// Communicating Units-------------------------------------------------------
      L     DB1715.DBD   10;
      L     DB1715.DBD  106;
      ==D   ;
      =     #ComCIP;

// emergency OK -------------------------------------------------------------
      A     DB1715.DBX   75.0; //General Emergency Stop OK
      =     #EStopOK;

NETWORK
TITLE =read other unit's data

      SET   ;

// ... General Unit ----------/

      CALL FC   563 (
           ActReq                   := M    101.0,
           PLCNo                    := DB1715.DBW   14,
           SourceUnitNo             := 99,
           IsTUnit                  := FALSE,
           DstComDRec               := DB1715.GEN,
           RET_VAL                  := #wRetVal);

// ... CIP Unit ------------- /
      L     DB1711.DBD   46; // Select
      L     L#0; // Off
      ==D   ;
      JC    ELS1;
      TAK   ;
      L     DB1915.DBD   10; // CIP 1
      ==D   ;
      JC    M101;
      TAK   ;
      L     DB1925.DBD   10; // CIP 2
      ==D   ;
      JC    M102;
      TAK   ;
      L     DB1935.DBD   10; // CIP 3
      ==D   ;
      JC    M103;
      JU    ELS1;
M101: NOP   0; // Do 1
      CALL FC   563 (
           ActReq                   := M    101.0,
           PLCNo                    := 3,
           SourceUnitNo             := 91,
           IsTUnit                  := FALSE,
           DstComDRec               := DB1715.CIP,
           RET_VAL                  := #wRetVal);

      JU    FIN1;
M102: NOP   0; // Do 2
      CALL FC   563 (
           ActReq                   := M    101.0,
           PLCNo                    := 3,
           SourceUnitNo             := 92,
           IsTUnit                  := FALSE,
           DstComDRec               := DB1715.CIP,
           RET_VAL                  := #wRetVal);

      JU    FIN1;
M103: NOP   0; // Do 3
      CALL FC   563 (
           ActReq                   := M    101.0,
           PLCNo                    := 3,
           SourceUnitNo             := 93,
           IsTUnit                  := FALSE,
           DstComDRec               := DB1715.CIP,
           RET_VAL                  := #wRetVal);

      JU    FIN1;
ELS1: L     0;
      T     #iTmp;
      CALL SFC   21 (
           BVAL                     := #iTmp,
           RET_VAL                  := #iRetVal,
           BLK                      := DB1715.CIP);

FIN1: NOP   0;

NETWORK
TITLE =remote start
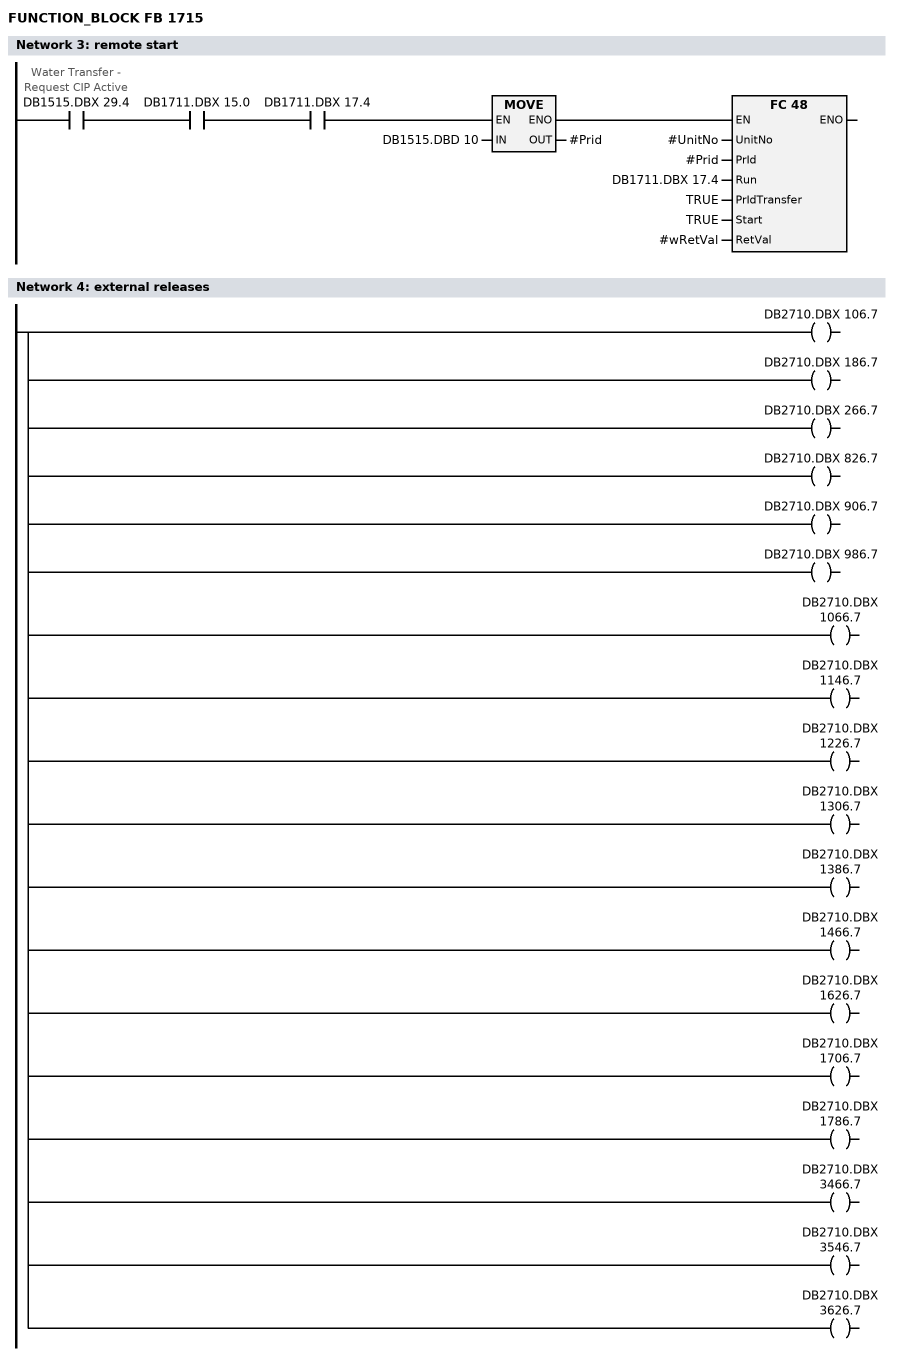

      SET   ;
      A     DB1515.DBX   29.4; // Water Transfer - Request CIP Active
      A     DB1711.DBX   15.0;
      A     DB1711.DBX   17.4;

      JCN   Strt;
      L     DB1515.DBD   10;
      T     #Prid;

      CALL FC    48 (
           UnitNo                   := #UnitNo,
           PrId                     := #Prid,
           Run                      := DB1711.DBX   17.4,
           PrIdTransfer             := TRUE,
           Start                    := TRUE,
           RetVal                   := #wRetVal);
Strt: NOP   0;
NETWORK
TITLE =external releases

      SET   ;
      =     DB2710.DBX  106.7;
      =     DB2710.DBX  186.7;
      =     DB2710.DBX  266.7;
      =     DB2710.DBX  826.7;
      =     DB2710.DBX  906.7;
      =     DB2710.DBX  986.7;
      =     DB2710.DBX 1066.7;
      =     DB2710.DBX 1146.7;
      =     DB2710.DBX 1226.7;
      =     DB2710.DBX 1306.7;
      =     DB2710.DBX 1386.7;
      =     DB2710.DBX 1466.7;
      =     DB2710.DBX 1626.7;
      =     DB2710.DBX 1706.7;
      =     DB2710.DBX 1786.7;
      =     DB2710.DBX 3466.7;
      =     DB2710.DBX 3546.7;
      =     DB2710.DBX 3626.7;
NETWORK
TITLE =write own unit data

      SET   ;

//-- CIP Communication ---------------------------------------
      AN    DB1711.DBX   15.0;
      AN    DB1711.DBX 1233.6; // CIP Active (Slave)
      A     #ComCIP;
      JCN   NCIP;
//Conductivity CIP Return
      L     DB1715.DBD  150;
      T     DB1711.DBD  626;

//Temperature CIP Return
      L     DB1715.DBD  146;
      T     DB1711.DBD  594;

//CIP Prerun Pump SP

      CALL FC    45 (
           SFM                      := DB1711.DBD  686,
           Indexes                  := #SFM36);


      L     0.000000e+000;
      A     #SFM36.I01;
      =     DB1715.DBX  171.7;
      JCN   pfc;
      L     DB1711.DBD  654;
pfc:  NOP   0;
      A     #SFM36.I02;
      =     DB1715.DBX  172.0;
      JCN   ppc;
      L     DB1711.DBD  670;
ppc:  NOP   0;
      A     #SFM36.I03;
      =     DB1715.DBX  171.6;
      JCN   pxc;
      L     DB1711.DBD  574;
pxc:  NOP   0;
      T     DB1715.DBD  182;

//CIP Return
      L     DB1711.DBD  558;
      T     DB1715.DBD  186;
      L     DB1715.DBD  138;
      T     DB1711.DBD  562;

//CIP Prerun
      L     DB1711.DBD  542;
      T     DB1715.DBD  190;
      L     DB1715.DBD  142;
      T     DB1711.DBD  546;

// Write Own Data to CIP
      L     DB1715.DBD   10;
      T     DB1715.DBD  154;

      L     DB1715.DBW   14;
      T     DB1715.DBW  158;

      L     DB1715.DBW   16;
      T     DB1715.DBW  160;

      L     DB1715.DBW   18;
      T     DB1715.DBW  162;

      L     DB1715.DBW   20;
      T     DB1715.DBW  164;

      L     DB1715.DBW   22;
      T     DB1715.DBW  166;

      A     DB1715.DBX   24.0;
      =     DB1715.DBX  168.0;

      A     DB1715.DBX   24.1;
      =     DB1715.DBX  168.1;

      A     DB1715.DBX   24.2;
      =     DB1715.DBX  168.2;

      A     DB1715.DBX   24.3;
      =     DB1715.DBX  168.3;

      A     DB1715.DBX   24.4;
      =     DB1715.DBX  168.4;

      A     DB1715.DBX   24.5;
      =     DB1715.DBX  168.5;

      A     DB1715.DBX   24.6;
      =     DB1715.DBX  168.6;

      A     DB1715.DBX   24.7;
      =     DB1715.DBX  168.7;

// Copy Data to CIP
      CALL SFC   20 (
           SRCBLK                   := DB1715.ToCIP,
           RET_VAL                  := #iRetVal,
           DSTBLK                   := DB1715.ToCIP);

NCIP: NOP   0;

//Empty Signal
//A     "U071SpID".SpI.Sig //!!!! Insert correct Empty Signal !!!
      CLR   ;
      =     DB1715.DBX   26.5;

//Full Signal
//A     "U071SpID".SpI.Sig //!!!! Insert correct Full Signal !!!
      CLR   ;
      =     DB1715.DBX   26.2;

//CIP Program Selected
      A     #CIP;
      =     DB1715.DBX   27.1;

// Emergency Stop
      A     #EStopOK; //If needed add or replace with own SpI
      =     DB1715.DBX   27.0; //Emergency Stop OK


NETWORK
TITLE =Signals to Filler / Mixer

// Watchdog
      A     M    100.7;
//    =     "F11_Watchdog"
//    =     "A11_Mixer_Watchdog"

      CLR   ;


END_FUNCTION_BLOCK

FUNCTION_BLOCK FB 1719
TITLE =U071: Packaging Plant 11
AUTHOR : Woermann
FAMILY : BOTEC_F1
NAME : Sim
VERSION : 0.1


VAR_TEMP
  CIP : BOOL ;	//CIP active
  xTmp : BOOL ;	//Temporary BOOL (free for general use)
  iTmp : INT ;	//Temporary INT (free for general use)
  rTmp : REAL ;	//Temporary REAL (free for general use)
  UnitNo : INT ;	//Unit Number
END_VAR
BEGIN
NETWORK
TITLE =General

      SET   ;
// get unit number ----------------------------------------------------------
      L     DB1710.DBW    0;
      T     #UnitNo;

// CIP ----------------------------------------------------------------------
      L     DB1711.DBD   54;
      L     0;
      <D    ;
      =     #CIP;

NETWORK
TITLE =Actuator

      A     DB1711.DBX   17.3;
      =     DB2710.DBX  105.3;
      =     DB2710.DBX  185.3;
      =     DB2710.DBX  265.3;
      =     DB2710.DBX  825.3;
      =     DB2710.DBX  905.3;
      =     DB2710.DBX  985.3;
      =     DB2710.DBX 1065.3;
      =     DB2710.DBX 1145.3;
      =     DB2710.DBX 1225.3;
      =     DB2710.DBX 1305.3;
      =     DB2710.DBX 1385.3;
      =     DB2710.DBX 1465.3;
      =     DB2710.DBX 1625.3;
      =     DB2710.DBX 1705.3;
      =     DB2710.DBX 1785.3;
      =     DB2710.DBX 3465.3;
      =     DB2710.DBX 3545.3;
      =     DB2710.DBX 3625.3;

NETWORK
TITLE =Special Input

      A     DB1711.DBX   17.3;
      =     DB2711.DBX  141.3;
      =     DB2711.DBX  201.3;
      =     DB2711.DBX  261.3;
      =     DB2711.DBX  321.3;
      =     DB2711.DBX  381.3;
      =     DB2711.DBX  681.3;
      =     DB2711.DBX  741.3;

NETWORK
TITLE =Counter

      A     DB1711.DBX   17.3;
      A     M    101.0;


      CLR   ;
NETWORK
TITLE =Analog Input

      A     DB1711.DBX   17.3;

NETWORK
TITLE =Universal Value

      A     DB1711.DBX   17.3;
//      =     "U071UnVD".unv001.Sim;
//      =     "U071UnVD".unv002.Sim;
//      =     "U071UnVD".unv003.Sim;
//      =     "U071UnVD".unv004.Sim;

NETWORK
TITLE =PID

      A     DB1711.DBX   17.3;

NETWORK
TITLE =Message

      A     DB1711.DBX   17.3;
//      =     "U071MsgD".msg001.Sim;
//      =     "U071MsgD".msg002.Sim;
//      =     "U071MsgD".msg003.Sim;

NETWORK
TITLE =VLT

      A     DB1711.DBX   17.3;

END_FUNCTION_BLOCK

FUNCTION_BLOCK FB 1725
TITLE =U072: Packaging Plant 12
FAMILY : BOTEC_F1
NAME : Comm
VERSION : 0.1


VAR_TEMP
  iRetVal : INT ;	//return value as integer
  wRetVal : WORD ;	//return value as word
  Run : BOOL ;	//Unit in "RUN" mode
  EStopOK : BOOL ;	//Emergency Stop OK
  CIP : BOOL ;	//CIP Program Selected
  ComCIP : BOOL ;	//Communication with CIP Active
  xTmp : BOOL ;	//Temporary BOOL (free for general use)
  iTmp : INT ;	//Temporary INT (free for general use)
  rTmp : REAL ;	//Temporary REAL (free for general use)
  dTmp : DINT ;	//Temporary DINT (free for general use)
  UnitNo : INT ;	//Unit Number
  EquipmentID : INT ;	//Equipment ID
  Prid : DINT ;	//Process ID
  SFM36 : STRUCT 	// CIP Pump Mode
   I00 : BOOL ;	// Off
   I01 : BOOL ;	// Flow
   I02 : BOOL ;	// Pressure
   I03 : BOOL ;	// Fix Speed
   I04 : BOOL ;
   I05 : BOOL ;
   I06 : BOOL ;
   I07 : BOOL ;
   I08 : BOOL ;
   I09 : BOOL ;
   I10 : BOOL ;
   I11 : BOOL ;
   I12 : BOOL ;
   I13 : BOOL ;
   I14 : BOOL ;
   I15 : BOOL ;
   I16 : BOOL ;
   I17 : BOOL ;
   I18 : BOOL ;
   I19 : BOOL ;
   I20 : BOOL ;
   I21 : BOOL ;
   I22 : BOOL ;
   I23 : BOOL ;
   I24 : BOOL ;
   I25 : BOOL ;
   I26 : BOOL ;
   I27 : BOOL ;
   I28 : BOOL ;
   I29 : BOOL ;
   I30 : BOOL ;
   I31 : BOOL ;
  END_STRUCT ;
END_VAR
BEGIN
NETWORK
TITLE =general

      SET   ;

// unit & equipment number ---------------------------------------------------
      L     DB1720.DBW    0;
      T     #UnitNo;

      L     DB1725.DBW   14;
      L     1000;
      *I    ;
      L     #UnitNo;
      +I    ;
      T     #EquipmentID;

// CIP ----------------------------------------------------------------------
      L     DB1725.DBW   18;
      L     0;
      <I    ;
      =     #CIP;

// Communicating Units-------------------------------------------------------
      L     DB1725.DBD   10;
      L     DB1725.DBD  106;
      ==D   ;
      =     #ComCIP;

// emergency OK -------------------------------------------------------------
      A     DB1725.DBX   75.0; //General Emergency Stop OK
      =     #EStopOK;

NETWORK
TITLE =read other unit's data

      SET   ;

// ... General Unit ----------/

      CALL FC   563 (
           ActReq                   := M    101.0,
           PLCNo                    := DB1725.DBW   14,
           SourceUnitNo             := 99,
           IsTUnit                  := FALSE,
           DstComDRec               := DB1725.GEN,
           RET_VAL                  := #wRetVal);


// ... CIP Unit ------------- /
      L     DB1721.DBD   46; // Select
      L     L#0; // Off
      ==D   ;
      JC    ELS1;
      TAK   ;
      L     DB1915.DBD   10; // CIP 1
      ==D   ;
      JC    M101;
      TAK   ;
      L     DB1925.DBD   10; // CIP 2
      ==D   ;
      JC    M102;
      TAK   ;
      L     DB1935.DBD   10; // CIP 3
      ==D   ;
      JC    M103;
      JU    ELS1;
M101: NOP   0; // Do 1
      CALL FC   563 (
           ActReq                   := M    101.0,
           PLCNo                    := 3,
           SourceUnitNo             := 91,
           IsTUnit                  := FALSE,
           DstComDRec               := DB1725.CIP,
           RET_VAL                  := #wRetVal);

      JU    FIN1;
M102: NOP   0; // Do 2
      CALL FC   563 (
           ActReq                   := M    101.0,
           PLCNo                    := 3,
           SourceUnitNo             := 92,
           IsTUnit                  := FALSE,
           DstComDRec               := DB1725.CIP,
           RET_VAL                  := #wRetVal);

      JU    FIN1;
M103: NOP   0; // Do 3
      CALL FC   563 (
           ActReq                   := M    101.0,
           PLCNo                    := 3,
           SourceUnitNo             := 93,
           IsTUnit                  := FALSE,
           DstComDRec               := DB1725.CIP,
           RET_VAL                  := #wRetVal);

      JU    FIN1;
ELS1: L     0;
      T     #iTmp;
      CALL SFC   21 (
           BVAL                     := #iTmp,
           RET_VAL                  := #iRetVal,
           BLK                      := DB1725.CIP);

FIN1: NOP   0;

NETWORK
TITLE =remote start
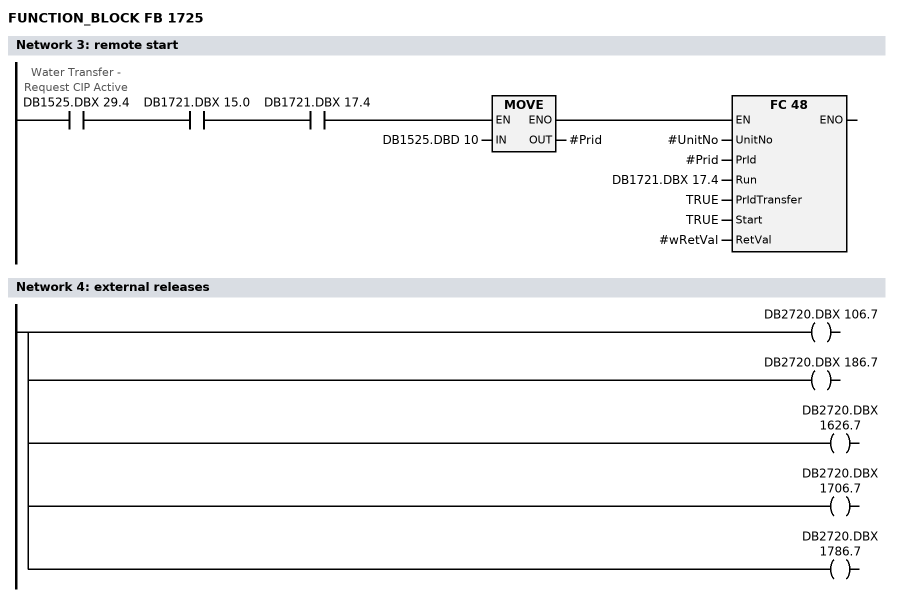

      SET   ;
      A     DB1525.DBX   29.4; // Water Transfer - Request CIP Active
      A     DB1721.DBX   15.0;
      A     DB1721.DBX   17.4;

      JCN   Strt;
      L     DB1525.DBD   10;
      T     #Prid;


      CALL FC    48 (
           UnitNo                   := #UnitNo,
           PrId                     := #Prid,
           Run                      := DB1721.DBX   17.4,
           PrIdTransfer             := TRUE,
           Start                    := TRUE,
           RetVal                   := #wRetVal);
Strt: NOP   0;
NETWORK
TITLE =external releases

      SET   ;
      =     DB2720.DBX  106.7;
      =     DB2720.DBX  186.7;
      =     DB2720.DBX 1626.7;
      =     DB2720.DBX 1706.7;
      =     DB2720.DBX 1786.7;
NETWORK
TITLE =write own unit data

      SET   ;

//-- CIP Communication ---------------------------------------
      AN    DB1721.DBX   15.0;
      AN    DB1721.DBX 1233.6; // CIP Active (Slave)
      A     #ComCIP;
      JCN   NCIP;
//Conductivity CIP Return
      L     DB1725.DBD  150;
      T     DB1721.DBD  626;

//Temperature CIP Return
      L     DB1725.DBD  146;
      T     DB1721.DBD  594;

//CIP Prerun Pump SP

      CALL FC    45 (
           SFM                      := DB1721.DBD  686,
           Indexes                  := #SFM36);


      L     0.000000e+000;
      A     #SFM36.I01;
      =     DB1725.DBX  171.7;
      JCN   pfc;
      L     DB1721.DBD  654;
pfc:  NOP   0;
      A     #SFM36.I02;
      =     DB1725.DBX  172.0;
      JCN   ppc;
      L     DB1721.DBD  670;
ppc:  NOP   0;
      A     #SFM36.I03;
      =     DB1725.DBX  171.6;
      JCN   pxc;
      L     DB1721.DBD  574;
pxc:  NOP   0;
      T     DB1725.DBD  182;

//CIP Return
      L     DB1721.DBD  558;
      T     DB1725.DBD  186;
      L     DB1725.DBD  138;
      T     DB1721.DBD  562;

//CIP Prerun
      L     DB1721.DBD  542;
      T     DB1725.DBD  190;
      L     DB1725.DBD  142;
      T     DB1721.DBD  546;

// Write Own Data to CIP
      L     DB1725.DBD   10;
      T     DB1725.DBD  154;

      L     DB1725.DBW   14;
      T     DB1725.DBW  158;

      L     DB1725.DBW   16;
      T     DB1725.DBW  160;

      L     DB1725.DBW   18;
      T     DB1725.DBW  162;

      L     DB1725.DBW   20;
      T     DB1725.DBW  164;

      L     DB1725.DBW   22;
      T     DB1725.DBW  166;

      A     DB1725.DBX   24.0;
      =     DB1725.DBX  168.0;

      A     DB1725.DBX   24.1;
      =     DB1725.DBX  168.1;

      A     DB1725.DBX   24.2;
      =     DB1725.DBX  168.2;

      A     DB1725.DBX   24.3;
      =     DB1725.DBX  168.3;

      A     DB1725.DBX   24.4;
      =     DB1725.DBX  168.4;

      A     DB1725.DBX   24.5;
      =     DB1725.DBX  168.5;

      A     DB1725.DBX   24.6;
      =     DB1725.DBX  168.6;

      A     DB1725.DBX   24.7;
      =     DB1725.DBX  168.7;

// Copy Data to CIP
      CALL SFC   20 (
           SRCBLK                   := DB1725.ToCIP,
           RET_VAL                  := #iRetVal,
           DSTBLK                   := DB1725.ToCIP);

NCIP: NOP   0;

//Empty Signal
//A     "U072SpID".SpI.Sig //!!!! Insert correct Empty Signal !!!
      CLR   ;
      =     DB1725.DBX   26.5;

//Full Signal
//A     "U072SpID".SpI.Sig //!!!! Insert correct Full Signal !!!
      CLR   ;
      =     DB1725.DBX   26.2;

//CIP Program Selected
      A     #CIP;
      =     DB1725.DBX   27.1;

// Emergency Stop
      A     #EStopOK; //If needed add or replace with own SpI
      =     DB1725.DBX   27.0; //Emergency Stop OK


NETWORK
TITLE =Signals to Filler / Mixer

// Watchdog
      A     M    100.7;
      =     Q    269.7;
      =     Q    271.6;


END_FUNCTION_BLOCK

FUNCTION_BLOCK FB 1729
TITLE =U072: Packaging Plant 12
AUTHOR : Woermann
FAMILY : BOTEC_F1
NAME : Sim
VERSION : 0.1


VAR_TEMP
  CIP : BOOL ;	//CIP active
  xTmp : BOOL ;	//Temporary BOOL (free for general use)
  iTmp : INT ;	//Temporary INT (free for general use)
  rTmp : REAL ;	//Temporary REAL (free for general use)
  UnitNo : INT ;	//Unit Number
END_VAR
BEGIN
NETWORK
TITLE =General

      SET   ;
// get unit number ----------------------------------------------------------
      L     DB1720.DBW    0;
      T     #UnitNo;

// CIP ----------------------------------------------------------------------
      L     DB1721.DBD   54;
      L     0;
      <D    ;
      =     #CIP;

NETWORK
TITLE =Actuator

      A     DB1721.DBX   17.3;
      =     DB2720.DBX  105.3;
      =     DB2720.DBX  185.3;
      =     DB2720.DBX 1625.3;
      =     DB2720.DBX 1705.3;
      =     DB2720.DBX 1785.3;

NETWORK
TITLE =Special Input

      A     DB1721.DBX   17.3;
      =     DB2721.DBX  441.3;
      =     DB2721.DBX  501.3;
      =     DB2721.DBX  561.3;
      =     DB2721.DBX  621.3;
      =     DB2721.DBX  681.3;
      =     DB2721.DBX  741.3;
      =     DB2721.DBX  801.3;

NETWORK
TITLE =Counter

      A     DB1721.DBX   17.3;
      A     M    101.0;


      CLR   ;
NETWORK
TITLE =Analog Input

      A     DB1721.DBX   17.3;

NETWORK
TITLE =Universal Value

      A     DB1721.DBX   17.3;
//      =     "U072UnVD".unv001.Sim;
//      =     "U072UnVD".unv002.Sim;
//      =     "U072UnVD".unv003.Sim;
//      =     "U072UnVD".unv004.Sim;

NETWORK
TITLE =PID

      A     DB1721.DBX   17.3;

NETWORK
TITLE =Message

      A     DB1721.DBX   17.3;
//      =     "U072MsgD".msg001.Sim;
//      =     "U072MsgD".msg002.Sim;
//      =     "U072MsgD".msg003.Sim;

NETWORK
TITLE =VLT

      A     DB1721.DBX   17.3;

END_FUNCTION_BLOCK

FUNCTION_BLOCK FB 1745
TITLE =U074: Packaging Plant 14
FAMILY : BOTEC_F1
NAME : Comm
VERSION : 0.1


VAR_TEMP
  iRetVal : INT ;	//return value as integer
  wRetVal : WORD ;	//return value as word
  Run : BOOL ;	//Unit in "RUN" mode
  EStopOK : BOOL ;	//Emergency Stop OK
  CIP : BOOL ;	//CIP Program Selected
  ComCIP : BOOL ;	//Communication with CIP Active
  xTmp : BOOL ;	//Temporary BOOL (free for general use)
  iTmp : INT ;	//Temporary INT (free for general use)
  rTmp : REAL ;	//Temporary REAL (free for general use)
  dTmp : DINT ;	//Temporary DINT (free for general use)
  UnitNo : INT ;	//Unit Number
  EquipmentID : INT ;	//Equipment ID
  Prid : DINT ;	//Process ID
  SFM36 : STRUCT 	// CIP Pump Mode
   I00 : BOOL ;	// Off
   I01 : BOOL ;	// Flow
   I02 : BOOL ;	// Pressure
   I03 : BOOL ;	// Fix Speed
   I04 : BOOL ;
   I05 : BOOL ;
   I06 : BOOL ;
   I07 : BOOL ;
   I08 : BOOL ;
   I09 : BOOL ;
   I10 : BOOL ;
   I11 : BOOL ;
   I12 : BOOL ;
   I13 : BOOL ;
   I14 : BOOL ;
   I15 : BOOL ;
   I16 : BOOL ;
   I17 : BOOL ;
   I18 : BOOL ;
   I19 : BOOL ;
   I20 : BOOL ;
   I21 : BOOL ;
   I22 : BOOL ;
   I23 : BOOL ;
   I24 : BOOL ;
   I25 : BOOL ;
   I26 : BOOL ;
   I27 : BOOL ;
   I28 : BOOL ;
   I29 : BOOL ;
   I30 : BOOL ;
   I31 : BOOL ;
  END_STRUCT ;
END_VAR
BEGIN
NETWORK
TITLE =general

      SET   ;

// unit & equipment number ---------------------------------------------------
      L     DB1740.DBW    0;
      T     #UnitNo;

      L     DB1745.DBW   14;
      L     1000;
      *I    ;
      L     #UnitNo;
      +I    ;
      T     #EquipmentID;

// CIP ----------------------------------------------------------------------
      L     DB1745.DBW   18;
      L     0;
      <I    ;
      =     #CIP;

// Communicating Units-------------------------------------------------------
      L     DB1745.DBD   10;
      L     DB1745.DBD  106;
      ==D   ;
      =     #ComCIP;

// emergency OK -------------------------------------------------------------
      A     DB1745.DBX   75.0; //General Emergency Stop OK
      =     #EStopOK;

NETWORK
TITLE =read other unit's data

      SET   ;

// ... General Unit ----------/

      CALL FC   563 (
           ActReq                   := M    101.0,
           PLCNo                    := DB1745.DBW   14,
           SourceUnitNo             := 99,
           IsTUnit                  := FALSE,
           DstComDRec               := DB1745.GEN,
           RET_VAL                  := #wRetVal);


// ... CIP Unit ------------- /
      L     DB1741.DBD   46; // Select
      L     L#0; // Off
      ==D   ;
      JC    ELS1;
      TAK   ;
      L     DB1915.DBD   10; // CIP 1
      ==D   ;
      JC    M101;
      TAK   ;
      L     DB1925.DBD   10; // CIP 2
      ==D   ;
      JC    M102;
      TAK   ;
      L     DB1935.DBD   10; // CIP 3
      ==D   ;
      JC    M103;
      JU    ELS1;
M101: NOP   0; // Do 1
      CALL FC   563 (
           ActReq                   := M    101.0,
           PLCNo                    := 3,
           SourceUnitNo             := 91,
           IsTUnit                  := FALSE,
           DstComDRec               := DB1745.CIP,
           RET_VAL                  := #wRetVal);

      JU    FIN1;
M102: NOP   0; // Do 2
      CALL FC   563 (
           ActReq                   := M    101.0,
           PLCNo                    := 3,
           SourceUnitNo             := 92,
           IsTUnit                  := FALSE,
           DstComDRec               := DB1745.CIP,
           RET_VAL                  := #wRetVal);

      JU    FIN1;
M103: NOP   0; // Do 3
      CALL FC   563 (
           ActReq                   := M    101.0,
           PLCNo                    := 3,
           SourceUnitNo             := 93,
           IsTUnit                  := FALSE,
           DstComDRec               := DB1745.CIP,
           RET_VAL                  := #wRetVal);

      JU    FIN1;
ELS1: L     0;
      T     #iTmp;
      CALL SFC   21 (
           BVAL                     := #iTmp,
           RET_VAL                  := #iRetVal,
           BLK                      := DB1745.CIP);

FIN1: NOP   0;

NETWORK
TITLE =remote start
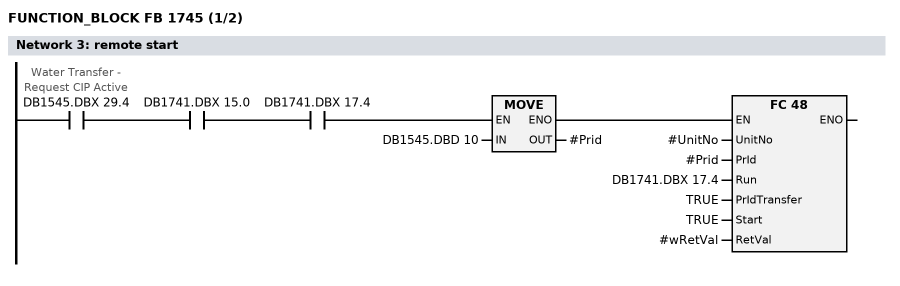

      SET   ;
      A     DB1545.DBX   29.4; // Water Transfer - Request CIP Active
      A     DB1741.DBX   15.0;
      A     DB1741.DBX   17.4;

      JCN   Strt;
      L     DB1545.DBD   10;
      T     #Prid;

      CALL FC    48 (
           UnitNo                   := #UnitNo,
           PrId                     := #Prid,
           Run                      := DB1741.DBX   17.4,
           PrIdTransfer             := TRUE,
           Start                    := TRUE,
           RetVal                   := #wRetVal);
Strt: NOP   0;
NETWORK
TITLE =external releases
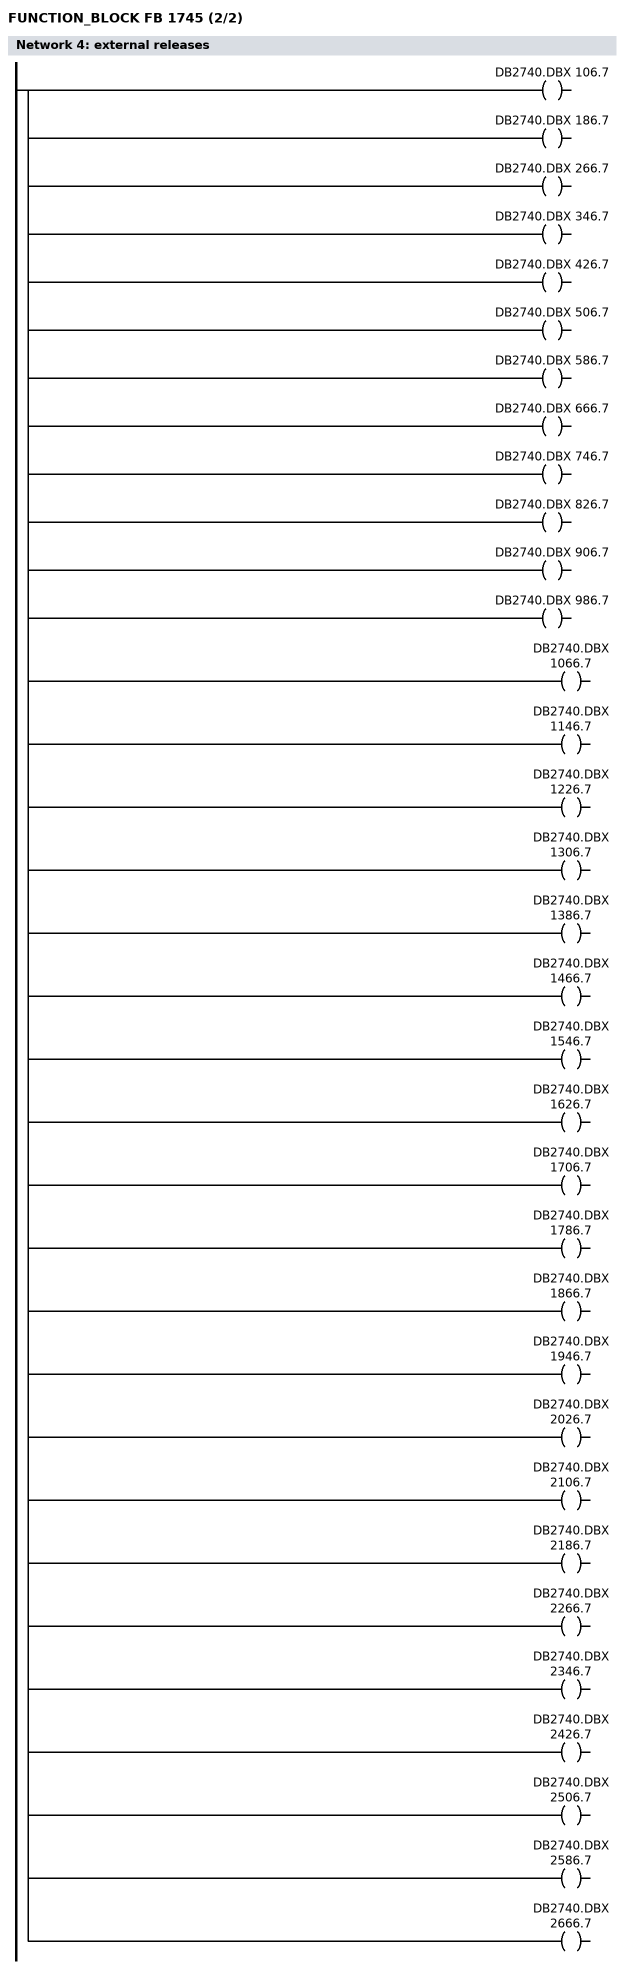

      SET   ;
      =     DB2740.DBX  106.7;
      =     DB2740.DBX  186.7;
      =     DB2740.DBX  266.7;
      =     DB2740.DBX  346.7;
      =     DB2740.DBX  426.7;
      =     DB2740.DBX  506.7;
      =     DB2740.DBX  586.7;
      =     DB2740.DBX  666.7;
      =     DB2740.DBX  746.7;
      =     DB2740.DBX  826.7;
      =     DB2740.DBX  906.7;
      =     DB2740.DBX  986.7;
      =     DB2740.DBX 1066.7;
      =     DB2740.DBX 1146.7;
      =     DB2740.DBX 1226.7;
      =     DB2740.DBX 1306.7;
      =     DB2740.DBX 1386.7;
      =     DB2740.DBX 1466.7;
      =     DB2740.DBX 1546.7;
      =     DB2740.DBX 1626.7;
      =     DB2740.DBX 1706.7;
      =     DB2740.DBX 1786.7;
      =     DB2740.DBX 1866.7;
      =     DB2740.DBX 1946.7;
      =     DB2740.DBX 2026.7;
      =     DB2740.DBX 2106.7;
      =     DB2740.DBX 2186.7;
      =     DB2740.DBX 2266.7;
      =     DB2740.DBX 2346.7;
      =     DB2740.DBX 2426.7;
      =     DB2740.DBX 2506.7;
      =     DB2740.DBX 2586.7;
      =     DB2740.DBX 2666.7;

NETWORK
TITLE =write own unit data

      SET   ;

//-- CIP Communication ---------------------------------------
      AN    DB1741.DBX   15.0;
//      AN "U074SeqD".Seq.PO.B30 // CIP Active (Slave)
      A     #ComCIP;
      JCN   NCIP;
//Conductivity CIP Return
      L     DB1745.DBD  150;
      T     DB1741.DBD  626;

//Temperature CIP Return
      L     DB1745.DBD  146;
      T     DB1741.DBD  594;

//CIP Prerun Pump SP

      CALL FC    45 (
           SFM                      := DB1741.DBD  686,
           Indexes                  := #SFM36);


      L     0.000000e+000;
      A     #SFM36.I01;
      =     DB1745.DBX  171.7;
      JCN   pfc;
      L     DB1741.DBD  654;
pfc:  NOP   0;
      A     #SFM36.I02;
      =     DB1745.DBX  172.0;
      JCN   ppc;
      L     DB1741.DBD  670;
ppc:  NOP   0;
      A     #SFM36.I03;
      =     DB1745.DBX  171.6;
      JCN   pxc;
      L     DB1741.DBD  574;
pxc:  NOP   0;
      T     DB1745.DBD  182;

//CIP Return
      L     DB1741.DBD  558;
      T     DB1745.DBD  186;
      L     DB1745.DBD  138;
      T     DB1741.DBD  562;

//CIP Prerun
      L     DB1741.DBD  542;
      T     DB1745.DBD  190;
      L     DB1745.DBD  142;
      T     DB1741.DBD  546;

// Write Own Data to CIP
      L     DB1745.DBD   10;
      T     DB1745.DBD  154;

      L     DB1745.DBW   14;
      T     DB1745.DBW  158;

      L     DB1745.DBW   16;
      T     DB1745.DBW  160;

      L     DB1745.DBW   18;
      T     DB1745.DBW  162;

      L     DB1745.DBW   20;
      T     DB1745.DBW  164;

      L     DB1745.DBW   22;
      T     DB1745.DBW  166;

      A     DB1745.DBX   24.0;
      =     DB1745.DBX  168.0;

      A     DB1745.DBX   24.1;
      =     DB1745.DBX  168.1;

      A     DB1745.DBX   24.2;
      =     DB1745.DBX  168.2;

      A     DB1745.DBX   24.3;
      =     DB1745.DBX  168.3;

      A     DB1745.DBX   24.4;
      =     DB1745.DBX  168.4;

      A     DB1745.DBX   24.5;
      =     DB1745.DBX  168.5;

      A     DB1745.DBX   24.6;
      =     DB1745.DBX  168.6;

      A     DB1745.DBX   24.7;
      =     DB1745.DBX  168.7;

// Copy Data to CIP
      CALL SFC   20 (
           SRCBLK                   := DB1745.ToCIP,
           RET_VAL                  := #iRetVal,
           DSTBLK                   := DB1745.ToCIP);

NCIP: NOP   0;

//Empty Signal
//A     "U074SpID".SpI.Sig //!!!! Insert correct Empty Signal !!!
      CLR   ;
      =     DB1745.DBX   26.5;

//Full Signal
//A     "U074SpID".SpI.Sig //!!!! Insert correct Full Signal !!!
      CLR   ;
      =     DB1745.DBX   26.2;

//CIP Program Selected
      A     #CIP;
      =     DB1745.DBX   27.1;

// Emergency Stop
      A     #EStopOK; //If needed add or replace with own SpI
      =     DB1745.DBX   27.0; //Emergency Stop OK


NETWORK
TITLE =Signals to Filler / Mixer
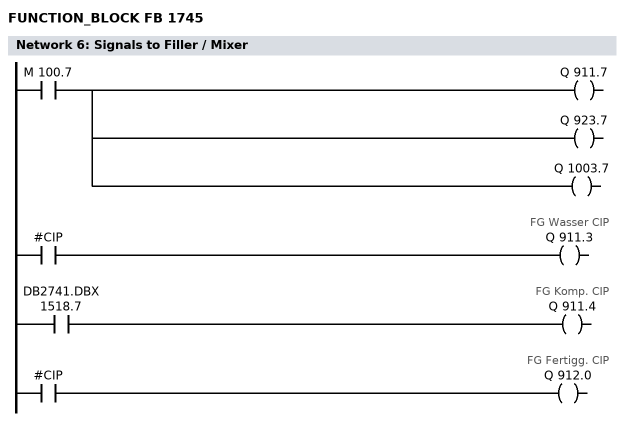

// Watchdog
      A     M    100.7;
      =     Q    911.7;
      =     Q    923.7;
      =     Q   1003.7;

// Panel

      A     #CIP;
      =     Q    911.3; // FG Wasser CIP
      A     DB2741.DBX 1518.7;
      =     Q    911.4; // FG Komp. CIP
      A     #CIP;
      =     Q    912.0; // FG Fertigg. CIP


END_FUNCTION_BLOCK

FUNCTION_BLOCK FB 1749
TITLE =U074: Packaging Plant 14
AUTHOR : Woermann
FAMILY : BOTEC_F1
NAME : Sim
VERSION : 0.1


VAR_TEMP
  CIP : BOOL ;	//CIP active
  xTmp : BOOL ;	//Temporary BOOL (free for general use)
  iTmp : INT ;	//Temporary INT (free for general use)
  rTmp : REAL ;	//Temporary REAL (free for general use)
  UnitNo : INT ;	//Unit Number
END_VAR
BEGIN
NETWORK
TITLE =General

      SET   ;
// get unit number ----------------------------------------------------------
      L     DB1740.DBW    0;
      T     #UnitNo;

// CIP ----------------------------------------------------------------------
      L     DB1741.DBD   54;
      L     0;
      <D    ;
      =     #CIP;

NETWORK
TITLE =Actuator

      A     DB1741.DBX   17.3;
      =     DB2740.DBX  105.3;
      =     DB2740.DBX  185.3;
      =     DB2740.DBX 1625.3;
      =     DB2740.DBX 1705.3;
      =     DB2740.DBX 1785.3;

NETWORK
TITLE =Special Input

      A     DB1741.DBX   17.3;
      =     DB2741.DBX 1581.3;
      =     DB2741.DBX 1641.3;

NETWORK
TITLE =Counter

      A     DB1741.DBX   17.3;
      A     M    101.0;


      CLR   ;
NETWORK
TITLE =Analog Input

      A     DB1741.DBX   17.3;

NETWORK
TITLE =Universal Value

      A     DB1741.DBX   17.3;
//      =     "U074UnVD".unv001.Sim;
//      =     "U074UnVD".unv002.Sim;
//      =     "U074UnVD".unv003.Sim;
//      =     "U074UnVD".unv004.Sim;

NETWORK
TITLE =PID

      A     DB1741.DBX   17.3;

NETWORK
TITLE =Message

      A     DB1741.DBX   17.3;
//      =     "U074MsgD".msg001.Sim;
//      =     "U074MsgD".msg002.Sim;
//      =     "U074MsgD".msg003.Sim;

NETWORK
TITLE =VLT

      A     DB1741.DBX   17.3;

END_FUNCTION_BLOCK

FUNCTION_BLOCK FB 1775
TITLE =U077: KZE Anlage  3
FAMILY : BOTEC_F1
NAME : U077Comm
VERSION : 0.1


VAR_TEMP
  iRetVal : INT ;	//return value as integer
  wRetVal : WORD ;	//return value as word
  Run : BOOL ;	//Unit in "RUN" mode
  EStopOK : BOOL ;	//Emergency Stop OK
  CIP : BOOL ;	//CIP Program Selected
  ComCIP : BOOL ;	//Communication with CIP Active
  xTmp : BOOL ;	//Temporary BOOL (free for general use)
  iTmp : INT ;	//Temporary INT (free for general use)
  rTmp : REAL ;	//Temporary REAL (free for general use)
  dTmp : DINT ;	//Temporary DINT (free for general use)
  UnitNo : INT ;	//Unit Number
  EquipmentID : INT ;	//Equipment ID
  Prid : DINT ;	//Process ID
  SFM36 : STRUCT 	// CIP Pump Mode
   I00 : BOOL ;	// Off
   I01 : BOOL ;	// Flow
   I02 : BOOL ;	// Pressure
   I03 : BOOL ;	// Fix Speed
   I04 : BOOL ;
   I05 : BOOL ;
   I06 : BOOL ;
   I07 : BOOL ;
   I08 : BOOL ;
   I09 : BOOL ;
   I10 : BOOL ;
   I11 : BOOL ;
   I12 : BOOL ;
   I13 : BOOL ;
   I14 : BOOL ;
   I15 : BOOL ;
   I16 : BOOL ;
   I17 : BOOL ;
   I18 : BOOL ;
   I19 : BOOL ;
   I20 : BOOL ;
   I21 : BOOL ;
   I22 : BOOL ;
   I23 : BOOL ;
   I24 : BOOL ;
   I25 : BOOL ;
   I26 : BOOL ;
   I27 : BOOL ;
   I28 : BOOL ;
   I29 : BOOL ;
   I30 : BOOL ;
   I31 : BOOL ;
  END_STRUCT ;
END_VAR
BEGIN
NETWORK
TITLE =general

      SET   ;

// unit & equipment number ---------------------------------------------------
      L     DB1770.DBW    0;
      T     #UnitNo;

      L     DB1775.DBW   14;
      L     1000;
      *I    ;
      L     #UnitNo;
      +I    ;
      T     #EquipmentID;

// CIP ----------------------------------------------------------------------
      L     DB1775.DBW   18;
      L     0;
      <I    ;
      =     #CIP;

// Communicating Units-------------------------------------------------------
      L     DB1775.DBD   10;
      L     DB1775.DBD  106;
      ==D   ;
      =     #ComCIP;

// emergency OK -------------------------------------------------------------
      A     DB1775.DBX   75.0; //General Emergency Stop OK
      CLR   ;
      =     #EStopOK;

NETWORK
TITLE =read other unit's data

      SET   ;

// ... General Unit ----------/

      CALL FC   563 (
           ActReq                   := M    101.0,
           PLCNo                    := 3,
           SourceUnitNo             := 99,
           IsTUnit                  := FALSE,
           DstComDRec               := DB1775.GEN,
           RET_VAL                  := #wRetVal);


NETWORK
TITLE =remote start

      SET   ;
// !!! insert correct condition of unit start !!!
      A     DB1771.DBX   15.0;
      A     DB1771.DBX   17.4;
      CLR   ;
      JCN   Strt;
      L     DB1775.DBD   10;
//L        L#-1;                            // Prid negative to start on its own
      T     #Prid;

      CALL FC    48 (
           UnitNo                   := #UnitNo,
           PrId                     := #Prid,
           Run                      := DB1771.DBX   17.4,
           PrIdTransfer             := TRUE,
           Start                    := TRUE,
           RetVal                   := #wRetVal);
Strt: NOP   0;
NETWORK
TITLE =external releases

      SET   ;

NETWORK
TITLE =write own unit data

      SET   ;

//-- CIP Communication ---------------------------------------
      AN    DB1771.DBX   15.0;
//      AN "U077SeqD".Seq.PO.B30 // CIP Active (Slave)
      A     #ComCIP;
      JCN   NCIP;
//Conductivity CIP Return
      L     DB1775.DBD  150;
      T     DB1771.DBD  626;

//Temperature CIP Return
      L     DB1775.DBD  146;
      T     DB1771.DBD  594;

//CIP Prerun Pump SP

      CALL FC    45 (
           SFM                      := DB1771.DBD  686,
           Indexes                  := #SFM36);


      L     0.000000e+000;
      A     #SFM36.I01;
      =     DB1775.DBX  171.7;
      JCN   pfc;
      L     DB1771.DBD  654;
pfc:  NOP   0;
      A     #SFM36.I02;
      =     DB1775.DBX  172.0;
      JCN   ppc;
      L     DB1771.DBD  670;
ppc:  NOP   0;
      A     #SFM36.I03;
      =     DB1775.DBX  171.6;
      JCN   pxc;
      L     DB1771.DBD  574;
pxc:  NOP   0;
      T     DB1775.DBD  182;

//CIP Return
      L     DB1771.DBD  558;
      T     DB1775.DBD  186;
      L     DB1775.DBD  138;
      T     DB1771.DBD  562;

//CIP Prerun
      L     DB1771.DBD  542;
      T     DB1775.DBD  190;
      L     DB1775.DBD  142;
      T     DB1771.DBD  546;

// Write Own Data to CIP
      L     DB1775.DBD   10;
      T     DB1775.DBD  154;

      L     DB1775.DBW   14;
      T     DB1775.DBW  158;

      L     DB1775.DBW   16;
      T     DB1775.DBW  160;

      L     DB1775.DBW   18;
      T     DB1775.DBW  162;

      L     DB1775.DBW   20;
      T     DB1775.DBW  164;

      L     DB1775.DBW   22;
      T     DB1775.DBW  166;

      A     DB1775.DBX   24.0;
      =     DB1775.DBX  168.0;

      A     DB1775.DBX   24.1;
      =     DB1775.DBX  168.1;

      A     DB1775.DBX   24.2;
      =     DB1775.DBX  168.2;

      A     DB1775.DBX   24.3;
      =     DB1775.DBX  168.3;

      A     DB1775.DBX   24.4;
      =     DB1775.DBX  168.4;

      A     DB1775.DBX   24.5;
      =     DB1775.DBX  168.5;

      A     DB1775.DBX   24.6;
      =     DB1775.DBX  168.6;

      A     DB1775.DBX   24.7;
      =     DB1775.DBX  168.7;

// Copy Data to CIP
      CALL SFC   20 (
           SRCBLK                   := DB1775.ToCIP,
           RET_VAL                  := #iRetVal,
           DSTBLK                   := DB1775.ToCIP);

NCIP: NOP   0;

//Empty Signal
//A     "U077SpID".SpI.Sig //!!!! Insert correct Empty Signal !!!
      CLR   ;
      =     DB1775.DBX   26.5;

//Full Signal
//A     "U077SpID".SpI.Sig //!!!! Insert correct Full Signal !!!
      CLR   ;
      =     DB1775.DBX   26.2;

//CIP Program Selected
      A     #CIP;
      =     DB1775.DBX   27.1;

// Emergency Stop
      A     #EStopOK; //If needed add or replace with own SpI
      =     DB1775.DBX   27.0; //Emergency Stop OK


NETWORK
TITLE = read from other unit data



END_FUNCTION_BLOCK

FUNCTION_BLOCK FB 1785
TITLE =U078: KZE Anlage  5
FAMILY : BOTEC_F1
NAME : U078Comm
VERSION : 0.1


VAR_TEMP
  iRetVal : INT ;	//return value as integer
  wRetVal : WORD ;	//return value as word
  Run : BOOL ;	//Unit in "RUN" mode
  EStopOK : BOOL ;	//Emergency Stop OK
  CIP : BOOL ;	//CIP Program Selected
  ComCIP : BOOL ;	//Communication with CIP Active
  xTmp : BOOL ;	//Temporary BOOL (free for general use)
  iTmp : INT ;	//Temporary INT (free for general use)
  rTmp : REAL ;	//Temporary REAL (free for general use)
  dTmp : DINT ;	//Temporary DINT (free for general use)
  UnitNo : INT ;	//Unit Number
  EquipmentID : INT ;	//Equipment ID
  Prid : DINT ;	//Process ID
  SFM36 : STRUCT 	// CIP Pump Mode
   I00 : BOOL ;	// Off
   I01 : BOOL ;	// Flow
   I02 : BOOL ;	// Pressure
   I03 : BOOL ;	// Fix Speed
   I04 : BOOL ;
   I05 : BOOL ;
   I06 : BOOL ;
   I07 : BOOL ;
   I08 : BOOL ;
   I09 : BOOL ;
   I10 : BOOL ;
   I11 : BOOL ;
   I12 : BOOL ;
   I13 : BOOL ;
   I14 : BOOL ;
   I15 : BOOL ;
   I16 : BOOL ;
   I17 : BOOL ;
   I18 : BOOL ;
   I19 : BOOL ;
   I20 : BOOL ;
   I21 : BOOL ;
   I22 : BOOL ;
   I23 : BOOL ;
   I24 : BOOL ;
   I25 : BOOL ;
   I26 : BOOL ;
   I27 : BOOL ;
   I28 : BOOL ;
   I29 : BOOL ;
   I30 : BOOL ;
   I31 : BOOL ;
  END_STRUCT ;
END_VAR
BEGIN
NETWORK
TITLE =general

      SET   ;

// unit & equipment number ---------------------------------------------------
      L     DB1780.DBW    0;
      T     #UnitNo;

      L     DB1785.DBW   14;
      L     1000;
      *I    ;
      L     #UnitNo;
      +I    ;
      T     #EquipmentID;

// CIP ----------------------------------------------------------------------
      L     DB1785.DBW   18;
      L     0;
      <I    ;
      =     #CIP;

// Communicating Units-------------------------------------------------------
      L     DB1785.DBD   10;
      L     DB1785.DBD  106;
      ==D   ;
      =     #ComCIP;

// emergency OK -------------------------------------------------------------
      A     DB1785.DBX   75.0; //General Emergency Stop OK
      =     #EStopOK;

NETWORK
TITLE =read other unit's data

      SET   ;

// ... General Unit ----------/

      CALL FC   563 (
           ActReq                   := M    101.0,
           PLCNo                    := 3,
           SourceUnitNo             := 99,
           IsTUnit                  := FALSE,
           DstComDRec               := DB1785.GEN,
           RET_VAL                  := #wRetVal);

NETWORK
TITLE =remote start

      SET   ;
// !!! insert correct condition of unit start !!!
      A     DB1781.DBX   15.0;
      A     DB1781.DBX   17.4;
      CLR   ;
      JCN   Strt;
      L     DB1785.DBD   10;
//L        L#-1;                            // Prid negative to start on its own
      T     #Prid;

      CALL FC    48 (
           UnitNo                   := #UnitNo,
           PrId                     := #Prid,
           Run                      := DB1781.DBX   17.4,
           PrIdTransfer             := TRUE,
           Start                    := TRUE,
           RetVal                   := #wRetVal);
Strt: NOP   0;
NETWORK
TITLE =external releases

      SET   ;
      =     DB2780.DBX  186.7;
      =     DB2780.DBX  266.7;
      =     DB2780.DBX  346.7;
      =     DB2780.DBX  426.7;
      =     DB2780.DBX  506.7;
      =     DB2780.DBX  586.7;
      =     DB2780.DBX  666.7;
      =     DB2780.DBX  986.7;
      =     DB2780.DBX 1066.7;
      =     DB2780.DBX 1146.7;
      =     DB2780.DBX 1226.7;
      =     DB2780.DBX 1306.7;
      =     DB2780.DBX 1386.7;
      =     DB2780.DBX 1626.7;
NETWORK
TITLE =write own unit data

      SET   ;

//-- CIP Communication ---------------------------------------
      AN    DB1781.DBX   15.0;
      AN    DB1781.DBX 1233.6; // CIP Active (Slave)
      A     #ComCIP;
      JCN   NCIP;
//Conductivity CIP Return
      L     DB1785.DBD  150;
      T     DB1781.DBD  626;

//Temperature CIP Return
      L     DB1785.DBD  146;
      T     DB1781.DBD  594;

//Temperature CIP Prerun
      L     DB1785.DBD  134;
      T     DB1781.DBD  690;

//CIP Prerun Pump SP

      CALL FC    45 (
           SFM                      := DB1781.DBD  686,
           Indexes                  := #SFM36);


      L     0.000000e+000;
      A     #SFM36.I01;
      =     DB1785.DBX  171.7;
      JCN   pfc;
      L     DB1781.DBD  654;
pfc:  NOP   0;
      A     #SFM36.I02;
      =     DB1785.DBX  172.0;
      JCN   ppc;
      L     DB1781.DBD  670;
ppc:  NOP   0;
      A     #SFM36.I03;
      =     DB1785.DBX  171.6;
      JCN   pxc;
      L     DB1781.DBD  574;
pxc:  NOP   0;
      T     DB1785.DBD  182;

// CIP Prerun Temperature
      L     DB1781.DBD  686;
      T     DB1785.DBD  182;

//CIP Return
      L     DB1781.DBD  558;
      T     DB1785.DBD  186;
      L     DB1785.DBD  138;
      T     DB1781.DBD  562;

//CIP Prerun
      L     DB1781.DBD  542;
      T     DB1785.DBD  190;
      L     DB1785.DBD  142;
      T     DB1781.DBD  546;

// Write Own Data to CIP
      L     DB1785.DBD   10;
      T     DB1785.DBD  154;

      L     DB1785.DBW   14;
      T     DB1785.DBW  158;

      L     DB1785.DBW   16;
      T     DB1785.DBW  160;

      L     DB1785.DBW   18;
      T     DB1785.DBW  162;

      L     DB1785.DBW   20;
      T     DB1785.DBW  164;

      L     DB1785.DBW   22;
      T     DB1785.DBW  166;

      A     DB1785.DBX   24.0;
      =     DB1785.DBX  168.0;

      A     DB1785.DBX   24.1;
      =     DB1785.DBX  168.1;

      A     DB1785.DBX   24.2;
      =     DB1785.DBX  168.2;

      A     DB1785.DBX   24.3;
      =     DB1785.DBX  168.3;

      A     DB1785.DBX   24.4;
      =     DB1785.DBX  168.4;

      A     DB1785.DBX   24.5;
      =     DB1785.DBX  168.5;

      A     DB1785.DBX   24.6;
      =     DB1785.DBX  168.6;

      A     DB1785.DBX   24.7;
      =     DB1785.DBX  168.7;

// Copy Data to CIP
      CALL SFC   20 (
           SRCBLK                   := DB1785.ToCIP,
           RET_VAL                  := #iRetVal,
           DSTBLK                   := DB1785.ToCIP);

NCIP: NOP   0;

//Empty Signal
//A     "U078SpID".SpI.Sig //!!!! Insert correct Empty Signal !!!
      CLR   ;
      =     DB1785.DBX   26.5;

//Full Signal
//A     "U078SpID".SpI.Sig //!!!! Insert correct Full Signal !!!
      CLR   ;
      =     DB1785.DBX   26.2;

//CIP Program Selected
      A     #CIP;
      =     DB1785.DBX   27.1;

// Emergency Stop
      A     #EStopOK; //If needed add or replace with own SpI
      =     DB1785.DBX   27.0; //Emergency Stop OK


NETWORK
TITLE = read from other unit data



// ... CIP / CIP Distribution ------------- /
      CALL FC   563 (
           ActReq                   := TRUE,
           PLCNo                    := 3,
           SourceUnitNo             := 91,
           IsTUnit                  := FALSE,
           DstComDRec               := DB1785.CIP,
           RET_VAL                  := #wRetVal);

      CALL FC   563 (
           ActReq                   := TRUE,
           PLCNo                    := 3,
           SourceUnitNo             := 94,
           IsTUnit                  := FALSE,
           DstComDRec               := DB1785.CIPDist,
           RET_VAL                  := #wRetVal);

      L     DB1781.DBD   46;
      L     DB1945.DBD   10;
      ==D   ;
      JCN   CIP1;
      CALL SFC   20 (
           SRCBLK                   := DB1785.ToCIP,
           RET_VAL                  := #iRetVal,
           DSTBLK                   := DB502.ToCIP1);

CIP1: NOP   0;

END_FUNCTION_BLOCK

FUNCTION_BLOCK FB 1795
TITLE =U079: KZE Anlage 14
FAMILY : BOTEC_F1
NAME : U079Comm
VERSION : 0.1


VAR_TEMP
  iRetVal : INT ;	//return value as integer
  wRetVal : WORD ;	//return value as word
  Run : BOOL ;	//Unit in "RUN" mode
  EStopOK : BOOL ;	//Emergency Stop OK
  CIP : BOOL ;	//CIP Program Selected
  ComCIP : BOOL ;	//Communication with CIP Active
  xTmp : BOOL ;	//Temporary BOOL (free for general use)
  iTmp : INT ;	//Temporary INT (free for general use)
  rTmp : REAL ;	//Temporary REAL (free for general use)
  dTmp : DINT ;	//Temporary DINT (free for general use)
  UnitNo : INT ;	//Unit Number
  EquipmentID : INT ;	//Equipment ID
  Prid : DINT ;	//Process ID
  SFM36 : STRUCT 	// CIP Pump Mode
   I00 : BOOL ;	// Off
   I01 : BOOL ;	// Flow
   I02 : BOOL ;	// Pressure
   I03 : BOOL ;	// Fix Speed
   I04 : BOOL ;
   I05 : BOOL ;
   I06 : BOOL ;
   I07 : BOOL ;
   I08 : BOOL ;
   I09 : BOOL ;
   I10 : BOOL ;
   I11 : BOOL ;
   I12 : BOOL ;
   I13 : BOOL ;
   I14 : BOOL ;
   I15 : BOOL ;
   I16 : BOOL ;
   I17 : BOOL ;
   I18 : BOOL ;
   I19 : BOOL ;
   I20 : BOOL ;
   I21 : BOOL ;
   I22 : BOOL ;
   I23 : BOOL ;
   I24 : BOOL ;
   I25 : BOOL ;
   I26 : BOOL ;
   I27 : BOOL ;
   I28 : BOOL ;
   I29 : BOOL ;
   I30 : BOOL ;
   I31 : BOOL ;
  END_STRUCT ;
END_VAR
BEGIN
NETWORK
TITLE =general

      SET   ;

// unit & equipment number ---------------------------------------------------
      L     DB1790.DBW    0;
      T     #UnitNo;

      L     DB1795.DBW   14;
      L     1000;
      *I    ;
      L     #UnitNo;
      +I    ;
      T     #EquipmentID;

// CIP ----------------------------------------------------------------------
      L     DB1795.DBW   18;
      L     0;
      <I    ;
      =     #CIP;

// Communicating Units-------------------------------------------------------
      L     DB1795.DBD   10;
      L     DB1795.DBD  106;
      ==D   ;
      =     #ComCIP;

// emergency OK -------------------------------------------------------------
      A     DB1795.DBX   75.0; //General Emergency Stop OK
      CLR   ;
      =     #EStopOK;

NETWORK
TITLE =read other unit's data

      SET   ;

// ... General Unit ----------/

      CALL FC   563 (
           ActReq                   := M    101.0,
           PLCNo                    := 3,
           SourceUnitNo             := 99,
           IsTUnit                  := FALSE,
           DstComDRec               := DB1795.GEN,
           RET_VAL                  := #wRetVal);


NETWORK
TITLE =remote start

      SET   ;
// !!! insert correct condition of unit start !!!
      A     DB1791.DBX   15.0;
      A     DB1791.DBX   17.4;
      CLR   ;
      JCN   Strt;
      L     DB1795.DBD   10;
//L        L#-1;                            // Prid negative to start on its own
      T     #Prid;

      CALL FC    48 (
           UnitNo                   := #UnitNo,
           PrId                     := #Prid,
           Run                      := DB1791.DBX   17.4,
           PrIdTransfer             := TRUE,
           Start                    := TRUE,
           RetVal                   := #wRetVal);
Strt: NOP   0;
NETWORK
TITLE =external releases

      SET   ;
      =     DB2790.DBX  186.7;
      =     DB2790.DBX  266.7;
      =     DB2790.DBX  426.7;
      =     DB2790.DBX  506.7;
      =     DB2790.DBX  586.7;
      =     DB2790.DBX  666.7;
      =     DB2790.DBX  986.7;
      =     DB2790.DBX 1066.7;
      =     DB2790.DBX 1146.7;
      =     DB2790.DBX 1226.7;
      =     DB2790.DBX 1306.7;
      =     DB2790.DBX 1386.7;
NETWORK
TITLE =write own unit data

      SET   ;

//-- CIP Communication ---------------------------------------
      AN    DB1791.DBX   15.0;
//      AN "U079SeqD".Seq.PO.B30 // CIP Active (Slave)
      A     #ComCIP;
      JCN   NCIP;
//Conductivity CIP Return
      L     DB1795.DBD  150;
      T     DB1791.DBD  626;

//Temperature CIP Return
      L     DB1795.DBD  146;
      T     DB1791.DBD  594;

//CIP Prerun Pump SP

      CALL FC    45 (
           SFM                      := DB1791.DBD  686,
           Indexes                  := #SFM36);


      L     0.000000e+000;
      A     #SFM36.I01;
      =     DB1795.DBX  171.7;
      JCN   pfc;
      L     DB1791.DBD  654;
pfc:  NOP   0;
      A     #SFM36.I02;
      =     DB1795.DBX  172.0;
      JCN   ppc;
      L     DB1791.DBD  670;
ppc:  NOP   0;
      A     #SFM36.I03;
      =     DB1795.DBX  171.6;
      JCN   pxc;
      L     DB1791.DBD  574;
pxc:  NOP   0;
      T     DB1795.DBD  182;

//CIP Return
      L     DB1791.DBD  558;
      T     DB1795.DBD  186;
      L     DB1795.DBD  138;
      T     DB1791.DBD  562;

//CIP Prerun
      L     DB1791.DBD  542;
      T     DB1795.DBD  190;
      L     DB1795.DBD  142;
      T     DB1791.DBD  546;

// Write Own Data to CIP
      L     DB1795.DBD   10;
      T     DB1795.DBD  154;

      L     DB1795.DBW   14;
      T     DB1795.DBW  158;

      L     DB1795.DBW   16;
      T     DB1795.DBW  160;

      L     DB1795.DBW   18;
      T     DB1795.DBW  162;

      L     DB1795.DBW   20;
      T     DB1795.DBW  164;

      L     DB1795.DBW   22;
      T     DB1795.DBW  166;

      A     DB1795.DBX   24.0;
      =     DB1795.DBX  168.0;

      A     DB1795.DBX   24.1;
      =     DB1795.DBX  168.1;

      A     DB1795.DBX   24.2;
      =     DB1795.DBX  168.2;

      A     DB1795.DBX   24.3;
      =     DB1795.DBX  168.3;

      A     DB1795.DBX   24.4;
      =     DB1795.DBX  168.4;

      A     DB1795.DBX   24.5;
      =     DB1795.DBX  168.5;

      A     DB1795.DBX   24.6;
      =     DB1795.DBX  168.6;

      A     DB1795.DBX   24.7;
      =     DB1795.DBX  168.7;

// Copy Data to CIP
      CALL SFC   20 (
           SRCBLK                   := DB1795.ToCIP,
           RET_VAL                  := #iRetVal,
           DSTBLK                   := DB1795.ToCIP);

NCIP: NOP   0;

//Empty Signal
//A     "U079SpID".SpI.Sig //!!!! Insert correct Empty Signal !!!
      CLR   ;
      =     DB1795.DBX   26.5;

//Full Signal
//A     "U079SpID".SpI.Sig //!!!! Insert correct Full Signal !!!
      CLR   ;
      =     DB1795.DBX   26.2;

//CIP Program Selected
      A     #CIP;
      =     DB1795.DBX   27.1;

// Emergency Stop
      A     #EStopOK; //If needed add or replace with own SpI
      =     DB1795.DBX   27.0; //Emergency Stop OK


NETWORK
TITLE = read from other unit data



END_FUNCTION_BLOCK

FUNCTION_BLOCK FB 1815
TITLE =U081: Caustic Tank
FAMILY : BOTEC_F1
NAME : Comm
VERSION : 0.1


VAR_TEMP
  iRetVal : INT ;	//return value as integer
  wRetVal : WORD ;	//return value as word
  Run : BOOL ;	//Unit in "RUN" mode
  EStopOK : BOOL ;	//Emergency Stop OK
  CIP : BOOL ;	//CIP Program Selected
  ComCIP : BOOL ;	//Communication with CIP Active
  xTmp : BOOL ;	//Temporary BOOL (free for general use)
  iTmp : INT ;	//Temporary INT (free for general use)
  rTmp : REAL ;	//Temporary REAL (free for general use)
  dTmp : DINT ;	//Temporary DINT (free for general use)
  UnitNo : INT ;	//Unit Number
  EquipmentID : INT ;	//Equipment ID
  Prid : DINT ;	//Process ID
  SFM36 : STRUCT 	// CIP Pump Mode
   I00 : BOOL ;	// Off
   I01 : BOOL ;	// Flow
   I02 : BOOL ;	// Pressure
   I03 : BOOL ;	// Fix Speed
   I04 : BOOL ;
   I05 : BOOL ;
   I06 : BOOL ;
   I07 : BOOL ;
   I08 : BOOL ;
   I09 : BOOL ;
   I10 : BOOL ;
   I11 : BOOL ;
   I12 : BOOL ;
   I13 : BOOL ;
   I14 : BOOL ;
   I15 : BOOL ;
   I16 : BOOL ;
   I17 : BOOL ;
   I18 : BOOL ;
   I19 : BOOL ;
   I20 : BOOL ;
   I21 : BOOL ;
   I22 : BOOL ;
   I23 : BOOL ;
   I24 : BOOL ;
   I25 : BOOL ;
   I26 : BOOL ;
   I27 : BOOL ;
   I28 : BOOL ;
   I29 : BOOL ;
   I30 : BOOL ;
   I31 : BOOL ;
  END_STRUCT ;
END_VAR
BEGIN
NETWORK
TITLE =general

      SET   ;

// unit & equipment number ---------------------------------------------------
      L     DB1810.DBW    0;
      T     #UnitNo;

      L     DB1815.DBW   14;
      L     1000;
      *I    ;
      L     #UnitNo;
      +I    ;
      T     #EquipmentID;

// CIP ----------------------------------------------------------------------
      L     DB1815.DBW   18;
      L     0;
      <I    ;
      =     #CIP;

// Communicating Units-------------------------------------------------------
      L     DB1815.DBD   10;
      L     DB1815.DBD  106;
      ==D   ;
      =     #ComCIP;

// emergency OK -------------------------------------------------------------
      A     DB1815.DBX   75.0; //General Emergency Stop OK
      =     #EStopOK;

NETWORK
TITLE =read other unit's data

      SET   ;

// ... General Unit ----------/

      CALL FC   563 (
           ActReq                   := M    101.0,
           PLCNo                    := DB1815.DBW   14,
           SourceUnitNo             := 99,
           IsTUnit                  := FALSE,
           DstComDRec               := DB1815.GEN,
           RET_VAL                  := #wRetVal);

NETWORK
TITLE =remote start

      SET   ;

      A     DB1811.DBX   15.0;
      A     DB1811.DBX   17.4;
      JCN   Strt;
      L     DB1815.DBD   10;
      L     L#-1; // Prid negative to start on its own
      T     #Prid;

      CALL FC    48 (
           UnitNo                   := #UnitNo,
           PrId                     := #Prid,
           Run                      := DB1811.DBX   17.4,
           PrIdTransfer             := TRUE,
           Start                    := TRUE,
           RetVal                   := #wRetVal);
Strt: NOP   0;
NETWORK
TITLE =external releases

      SET   ;
      =     DB2810.DBX  106.7;
      =     DB2810.DBX  186.7;
      =     DB2810.DBX  266.7;
      =     DB2810.DBX  346.7;
      =     DB2810.DBX  426.7;
      =     DB2810.DBX  506.7;
      =     DB2810.DBX  586.7;
      =     DB2810.DBX  666.7;
      =     DB2810.DBX  746.7;
NETWORK
TITLE =write own unit data

      SET   ;

//-- CIP Communication ---------------------------------------
      AN    DB1811.DBX   15.0;
//      AN "U081SeqD".Seq.PO.B30 // CIP Active (Slave)
      A     #ComCIP;
      JCN   NCIP;
//Conductivity CIP Return
      L     DB1815.DBD  150;
      T     DB1811.DBD  626;

//Temperature CIP Return
      L     DB1815.DBD  146;
      T     DB1811.DBD  594;

//CIP Prerun Pump SP

      CALL FC    45 (
           SFM                      := DB1811.DBD  686,
           Indexes                  := #SFM36);


      L     0.000000e+000;
      A     #SFM36.I01;
      =     DB1815.DBX  171.7;
      JCN   pfc;
      L     DB1811.DBD  654;
pfc:  NOP   0;
      A     #SFM36.I02;
      =     DB1815.DBX  172.0;
      JCN   ppc;
      L     DB1811.DBD  670;
ppc:  NOP   0;
      A     #SFM36.I03;
      =     DB1815.DBX  171.6;
      JCN   pxc;
      L     DB1811.DBD  574;
pxc:  NOP   0;
      T     DB1815.DBD  182;

//CIP Return
      L     DB1811.DBD  558;
      T     DB1815.DBD  186;
      L     DB1815.DBD  138;
      T     DB1811.DBD  562;

//CIP Prerun
      L     DB1811.DBD  542;
      T     DB1815.DBD  190;
      L     DB1815.DBD  142;
      T     DB1811.DBD  546;

// Write Own Data to CIP
      L     DB1815.DBD   10;
      T     DB1815.DBD  154;

      L     DB1815.DBW   14;
      T     DB1815.DBW  158;

      L     DB1815.DBW   16;
      T     DB1815.DBW  160;

      L     DB1815.DBW   18;
      T     DB1815.DBW  162;

      L     DB1815.DBW   20;
      T     DB1815.DBW  164;

      L     DB1815.DBW   22;
      T     DB1815.DBW  166;

      A     DB1815.DBX   24.0;
      =     DB1815.DBX  168.0;

      A     DB1815.DBX   24.1;
      =     DB1815.DBX  168.1;

      A     DB1815.DBX   24.2;
      =     DB1815.DBX  168.2;

      A     DB1815.DBX   24.3;
      =     DB1815.DBX  168.3;

      A     DB1815.DBX   24.4;
      =     DB1815.DBX  168.4;

      A     DB1815.DBX   24.5;
      =     DB1815.DBX  168.5;

      A     DB1815.DBX   24.6;
      =     DB1815.DBX  168.6;

      A     DB1815.DBX   24.7;
      =     DB1815.DBX  168.7;

// Copy Data to CIP
      CALL SFC   20 (
           SRCBLK                   := DB1815.ToCIP,
           RET_VAL                  := #iRetVal,
           DSTBLK                   := DB1815.ToCIP);

NCIP: NOP   0;

//Empty Signal
      A     DB2811.DBX   78.7;
      =     DB1815.DBX   26.5;

//Full Signal
      AN    DB2811.DBX  138.7;
      O     DB2813.DBX  138.4;
      =     DB1815.DBX   26.2;

//CIP Program Selected
      A     #CIP;
      =     DB1815.DBX   27.1;

// Emergency Stop
      A     #EStopOK; //If needed add or replace with own SpI
      =     DB1815.DBX   27.0; //Emergency Stop OK


NETWORK
TITLE = read from other unit data



END_FUNCTION_BLOCK

FUNCTION_BLOCK FB 1819
TITLE =U081: Caustic Tank
AUTHOR : Woermann
FAMILY : BOTEC_F1
NAME : Sim
VERSION : 0.1


VAR_TEMP
  CIP : BOOL ;	//CIP active
  xTmp : BOOL ;	//Temporary BOOL (free for general use)
  iTmp : INT ;	//Temporary INT (free for general use)
  rTmp : REAL ;	//Temporary REAL (free for general use)
  UnitNo : INT ;	//Unit Number
END_VAR
BEGIN
NETWORK
TITLE =General

      SET   ;
// get unit number ----------------------------------------------------------
      L     DB1810.DBW    0;
      T     #UnitNo;

// CIP ----------------------------------------------------------------------
      L     DB1811.DBD   54;
      L     0;
      <D    ;
      =     #CIP;

NETWORK
TITLE =Actuator

      A     DB1811.DBX   17.3;
      =     DB2810.DBX  105.3;
      =     DB2810.DBX  185.3;
      =     DB2810.DBX  265.3;
      =     DB2810.DBX  345.3;
      =     DB2810.DBX  425.3;
      =     DB2810.DBX  505.3;
      =     DB2810.DBX  585.3;
      =     DB2810.DBX  665.3;
      =     DB2810.DBX  745.3;

NETWORK
TITLE =Special Input

      A     DB1811.DBX   17.3;
      =     DB2811.DBX   81.3;
      =     DB2811.DBX  141.3;
      =     DB2811.DBX  201.3;
      =     DB2811.DBX  261.3;
      =     DB2811.DBX  321.3;
      =     DB2811.DBX  441.3;
      =     DB2811.DBX  501.3;

NETWORK
TITLE =Counter

      A     DB1811.DBX   17.3;
      A     M    101.0;


      CLR   ;
NETWORK
TITLE =Analog Input

      A     DB1811.DBX   17.3;
      =     DB2813.DBX  141.3;
      =     DB2813.DBX  261.3;

NETWORK
TITLE =Universal Value

      A     DB1811.DBX   17.3;
//      =     "U081UnVD".unv001.Sim;
//      =     "U081UnVD".unv002.Sim;

NETWORK
TITLE =PID

      A     DB1811.DBX   17.3;

NETWORK
TITLE =Message

      A     DB1811.DBX   17.3;
//      =     "U081MsgD".msg001.Sim;
//      =     "U081MsgD".msg002.Sim;

NETWORK
TITLE =VLT

      A     DB1811.DBX   17.3;

END_FUNCTION_BLOCK

FUNCTION_BLOCK FB 1825
TITLE =U082: Acid Tank
FAMILY : BOTEC_F1
NAME : Comm
VERSION : 0.1


VAR_TEMP
  iRetVal : INT ;	//return value as integer
  wRetVal : WORD ;	//return value as word
  Run : BOOL ;	//Unit in "RUN" mode
  EStopOK : BOOL ;	//Emergency Stop OK
  CIP : BOOL ;	//CIP Program Selected
  ComCIP : BOOL ;	//Communication with CIP Active
  xTmp : BOOL ;	//Temporary BOOL (free for general use)
  iTmp : INT ;	//Temporary INT (free for general use)
  rTmp : REAL ;	//Temporary REAL (free for general use)
  dTmp : DINT ;	//Temporary DINT (free for general use)
  UnitNo : INT ;	//Unit Number
  EquipmentID : INT ;	//Equipment ID
  Prid : DINT ;	//Process ID
  SFM36 : STRUCT 	// CIP Pump Mode
   I00 : BOOL ;	// Off
   I01 : BOOL ;	// Flow
   I02 : BOOL ;	// Pressure
   I03 : BOOL ;	// Fix Speed
   I04 : BOOL ;
   I05 : BOOL ;
   I06 : BOOL ;
   I07 : BOOL ;
   I08 : BOOL ;
   I09 : BOOL ;
   I10 : BOOL ;
   I11 : BOOL ;
   I12 : BOOL ;
   I13 : BOOL ;
   I14 : BOOL ;
   I15 : BOOL ;
   I16 : BOOL ;
   I17 : BOOL ;
   I18 : BOOL ;
   I19 : BOOL ;
   I20 : BOOL ;
   I21 : BOOL ;
   I22 : BOOL ;
   I23 : BOOL ;
   I24 : BOOL ;
   I25 : BOOL ;
   I26 : BOOL ;
   I27 : BOOL ;
   I28 : BOOL ;
   I29 : BOOL ;
   I30 : BOOL ;
   I31 : BOOL ;
  END_STRUCT ;
END_VAR
BEGIN
NETWORK
TITLE =general

      SET   ;

// unit & equipment number ---------------------------------------------------
      L     DB1820.DBW    0;
      T     #UnitNo;

      L     DB1825.DBW   14;
      L     1000;
      *I    ;
      L     #UnitNo;
      +I    ;
      T     #EquipmentID;

// CIP ----------------------------------------------------------------------
      L     DB1825.DBW   18;
      L     0;
      <I    ;
      =     #CIP;

// Communicating Units-------------------------------------------------------
      L     DB1825.DBD   10;
      L     DB1825.DBD  106;
      ==D   ;
      =     #ComCIP;

// emergency OK -------------------------------------------------------------
      A     DB1825.DBX   75.0; //General Emergency Stop OK
      =     #EStopOK;

NETWORK
TITLE =read other unit's data

      SET   ;

// ... General Unit ----------/

      CALL FC   563 (
           ActReq                   := M    101.0,
           PLCNo                    := DB1825.DBW   14,
           SourceUnitNo             := 99,
           IsTUnit                  := FALSE,
           DstComDRec               := DB1825.GEN,
           RET_VAL                  := #wRetVal);

NETWORK
TITLE =remote start

      SET   ;

      A     DB1821.DBX   15.0;
      A     DB1821.DBX   17.4;
      JCN   Strt;
      L     DB1825.DBD   10;
      L     L#-1; // Prid negative to start on its own
      T     #Prid;

      CALL FC    48 (
           UnitNo                   := #UnitNo,
           PrId                     := #Prid,
           Run                      := DB1821.DBX   17.4,
           PrIdTransfer             := TRUE,
           Start                    := TRUE,
           RetVal                   := #wRetVal);
Strt: NOP   0;
NETWORK
TITLE =external releases

      SET   ;
      =     DB2820.DBX  106.7;
      =     DB2820.DBX  186.7;
      =     DB2820.DBX  346.7;
      =     DB2820.DBX  426.7;
      =     DB2820.DBX  586.7;
      =     DB2820.DBX  666.7;
      =     DB2820.DBX  746.7;
NETWORK
TITLE =write own unit data

      SET   ;

//-- CIP Communication ---------------------------------------
      AN    DB1821.DBX   15.0;
//      AN "U082SeqD".Seq.PO.B30 // CIP Active (Slave)
      A     #ComCIP;
      JCN   NCIP;
//Conductivity CIP Return
      L     DB1825.DBD  150;
      T     DB1821.DBD  626;

//Temperature CIP Return
      L     DB1825.DBD  146;
      T     DB1821.DBD  594;

//CIP Prerun Pump SP

      CALL FC    45 (
           SFM                      := DB1821.DBD  686,
           Indexes                  := #SFM36);


      L     0.000000e+000;
      A     #SFM36.I01;
      =     DB1825.DBX  171.7;
      JCN   pfc;
      L     DB1821.DBD  654;
pfc:  NOP   0;
      A     #SFM36.I02;
      =     DB1825.DBX  172.0;
      JCN   ppc;
      L     DB1821.DBD  670;
ppc:  NOP   0;
      A     #SFM36.I03;
      =     DB1825.DBX  171.6;
      JCN   pxc;
      L     DB1821.DBD  574;
pxc:  NOP   0;
      T     DB1825.DBD  182;

//CIP Return
      L     DB1821.DBD  558;
      T     DB1825.DBD  186;
      L     DB1825.DBD  138;
      T     DB1821.DBD  562;

//CIP Prerun
      L     DB1821.DBD  542;
      T     DB1825.DBD  190;
      L     DB1825.DBD  142;
      T     DB1821.DBD  546;

// Write Own Data to CIP
      L     DB1825.DBD   10;
      T     DB1825.DBD  154;

      L     DB1825.DBW   14;
      T     DB1825.DBW  158;

      L     DB1825.DBW   16;
      T     DB1825.DBW  160;

      L     DB1825.DBW   18;
      T     DB1825.DBW  162;

      L     DB1825.DBW   20;
      T     DB1825.DBW  164;

      L     DB1825.DBW   22;
      T     DB1825.DBW  166;

      A     DB1825.DBX   24.0;
      =     DB1825.DBX  168.0;

      A     DB1825.DBX   24.1;
      =     DB1825.DBX  168.1;

      A     DB1825.DBX   24.2;
      =     DB1825.DBX  168.2;

      A     DB1825.DBX   24.3;
      =     DB1825.DBX  168.3;

      A     DB1825.DBX   24.4;
      =     DB1825.DBX  168.4;

      A     DB1825.DBX   24.5;
      =     DB1825.DBX  168.5;

      A     DB1825.DBX   24.6;
      =     DB1825.DBX  168.6;

      A     DB1825.DBX   24.7;
      =     DB1825.DBX  168.7;

// Copy Data to CIP
      CALL SFC   20 (
           SRCBLK                   := DB1825.ToCIP,
           RET_VAL                  := #iRetVal,
           DSTBLK                   := DB1825.ToCIP);

NCIP: NOP   0;

//Empty Signal
      A     DB2821.DBX   78.7;
      =     DB1825.DBX   26.5;

//Full Signal
      AN    DB2821.DBX  138.7;
      O     DB2823.DBX  138.4;
      =     DB1825.DBX   26.2;

//CIP Program Selected
      A     #CIP;
      =     DB1825.DBX   27.1;

// Emergency Stop
      A     #EStopOK; //If needed add or replace with own SpI
      =     DB1825.DBX   27.0; //Emergency Stop OK


NETWORK
TITLE = read from other unit data



END_FUNCTION_BLOCK

FUNCTION_BLOCK FB 1829
TITLE =U082: Acid Tank
AUTHOR : Woermann
FAMILY : BOTEC_F1
NAME : Sim
VERSION : 0.1


VAR_TEMP
  CIP : BOOL ;	//CIP active
  xTmp : BOOL ;	//Temporary BOOL (free for general use)
  iTmp : INT ;	//Temporary INT (free for general use)
  rTmp : REAL ;	//Temporary REAL (free for general use)
  UnitNo : INT ;	//Unit Number
END_VAR
BEGIN
NETWORK
TITLE =General

      SET   ;
// get unit number ----------------------------------------------------------
      L     DB1820.DBW    0;
      T     #UnitNo;

// CIP ----------------------------------------------------------------------
      L     DB1821.DBD   54;
      L     0;
      <D    ;
      =     #CIP;

NETWORK
TITLE =Actuator

      A     DB1821.DBX   17.3;
      =     DB2820.DBX  105.3;
      =     DB2820.DBX  185.3;
      =     DB2820.DBX  345.3;
      =     DB2820.DBX  425.3;
      =     DB2820.DBX  585.3;
      =     DB2820.DBX  665.3;
      =     DB2820.DBX  745.3;

NETWORK
TITLE =Special Input

      A     DB1821.DBX   17.3;
      =     DB2821.DBX   81.3;
      =     DB2821.DBX  141.3;
      =     DB2821.DBX  201.3;
      =     DB2821.DBX  261.3;
      =     DB2821.DBX  441.3;
      =     DB2821.DBX  501.3;

NETWORK
TITLE =Counter

      A     DB1821.DBX   17.3;
      A     M    101.0;


      CLR   ;
NETWORK
TITLE =Analog Input

      A     DB1821.DBX   17.3;
      =     DB2823.DBX  141.3;
      =     DB2823.DBX  261.3;

NETWORK
TITLE =Universal Value

      A     DB1821.DBX   17.3;
//      =     "U082UnVD".unv001.Sim;
//      =     "U082UnVD".unv002.Sim;

NETWORK
TITLE =PID

      A     DB1821.DBX   17.3;

NETWORK
TITLE =Message

      A     DB1821.DBX   17.3;
//      =     "U082MsgD".msg001.Sim;
//      =     "U082MsgD".msg002.Sim;

NETWORK
TITLE =VLT

      A     DB1821.DBX   17.3;

END_FUNCTION_BLOCK

FUNCTION_BLOCK FB 1835
TITLE =U083: Hot Water Tank
FAMILY : BOTEC_F1
NAME : Comm
VERSION : 0.1


VAR_TEMP
  iRetVal : INT ;	//return value as integer
  wRetVal : WORD ;	//return value as word
  Run : BOOL ;	//Unit in "RUN" mode
  EStopOK : BOOL ;	//Emergency Stop OK
  CIP : BOOL ;	//CIP Program Selected
  ComCIP : BOOL ;	//Communication with CIP Active
  xTmp : BOOL ;	//Temporary BOOL (free for general use)
  iTmp : INT ;	//Temporary INT (free for general use)
  rTmp : REAL ;	//Temporary REAL (free for general use)
  dTmp : DINT ;	//Temporary DINT (free for general use)
  UnitNo : INT ;	//Unit Number
  EquipmentID : INT ;	//Equipment ID
  Prid : DINT ;	//Process ID
  SFM36 : STRUCT 	// CIP Pump Mode
   I00 : BOOL ;	// Off
   I01 : BOOL ;	// Flow
   I02 : BOOL ;	// Pressure
   I03 : BOOL ;	// Fix Speed
   I04 : BOOL ;
   I05 : BOOL ;
   I06 : BOOL ;
   I07 : BOOL ;
   I08 : BOOL ;
   I09 : BOOL ;
   I10 : BOOL ;
   I11 : BOOL ;
   I12 : BOOL ;
   I13 : BOOL ;
   I14 : BOOL ;
   I15 : BOOL ;
   I16 : BOOL ;
   I17 : BOOL ;
   I18 : BOOL ;
   I19 : BOOL ;
   I20 : BOOL ;
   I21 : BOOL ;
   I22 : BOOL ;
   I23 : BOOL ;
   I24 : BOOL ;
   I25 : BOOL ;
   I26 : BOOL ;
   I27 : BOOL ;
   I28 : BOOL ;
   I29 : BOOL ;
   I30 : BOOL ;
   I31 : BOOL ;
  END_STRUCT ;
END_VAR
BEGIN
NETWORK
TITLE =general

      SET   ;

// unit & equipment number ---------------------------------------------------
      L     DB1830.DBW    0;
      T     #UnitNo;

      L     DB1835.DBW   14;
      L     1000;
      *I    ;
      L     #UnitNo;
      +I    ;
      T     #EquipmentID;

// CIP ----------------------------------------------------------------------
      L     DB1835.DBW   18;
      L     0;
      <I    ;
      =     #CIP;

// Communicating Units-------------------------------------------------------
      L     DB1835.DBD   10;
      L     DB1835.DBD  106;
      ==D   ;
      =     #ComCIP;

// emergency OK -------------------------------------------------------------
      A     DB1835.DBX   75.0; //General Emergency Stop OK
      =     #EStopOK;

NETWORK
TITLE =read other unit's data

      SET   ;

// ... General Unit ----------/

      CALL FC   563 (
           ActReq                   := M    101.0,
           PLCNo                    := DB1835.DBW   14,
           SourceUnitNo             := 99,
           IsTUnit                  := FALSE,
           DstComDRec               := DB1835.GEN,
           RET_VAL                  := #wRetVal);

NETWORK
TITLE =remote start

      SET   ;

      A     DB1831.DBX   15.0;
      A     DB1831.DBX   17.4;
      JCN   Strt;
      L     DB1835.DBD   10;
      L     L#-1; // Prid negative to start on its own
      T     #Prid;

      CALL FC    48 (
           UnitNo                   := #UnitNo,
           PrId                     := #Prid,
           Run                      := DB1831.DBX   17.4,
           PrIdTransfer             := TRUE,
           Start                    := TRUE,
           RetVal                   := #wRetVal);
Strt: NOP   0;
NETWORK
TITLE =external releases

      SET   ;
      =     DB2830.DBX  106.7;
      =     DB2830.DBX  186.7;
      =     DB2830.DBX  266.7;
      =     DB2830.DBX  346.7;
      =     DB2830.DBX  426.7;
      =     DB2830.DBX  586.7;
      =     DB2830.DBX  746.7;
      =     DB2830.DBX  826.7;
      =     DB2830.DBX  906.7;
      =     DB2830.DBX  986.7;
      =     DB2830.DBX 1066.7;
NETWORK
TITLE =write own unit data

      SET   ;

//-- CIP Communication ---------------------------------------
      AN    DB1831.DBX   15.0;
//      AN "U083SeqD".Seq.PO.B30 // CIP Active (Slave)
      A     #ComCIP;
      JCN   NCIP;
//Conductivity CIP Return
      L     DB1835.DBD  150;
      T     DB1831.DBD  626;

//Temperature CIP Return
      L     DB1835.DBD  146;
      T     DB1831.DBD  594;

//CIP Prerun Pump SP

      CALL FC    45 (
           SFM                      := DB1831.DBD  686,
           Indexes                  := #SFM36);


      L     0.000000e+000;
      A     #SFM36.I01;
      =     DB1835.DBX  171.7;
      JCN   pfc;
      L     DB1831.DBD  654;
pfc:  NOP   0;
      A     #SFM36.I02;
      =     DB1835.DBX  172.0;
      JCN   ppc;
      L     DB1831.DBD  670;
ppc:  NOP   0;
      A     #SFM36.I03;
      =     DB1835.DBX  171.6;
      JCN   pxc;
      L     DB1831.DBD  574;
pxc:  NOP   0;
      T     DB1835.DBD  182;

//CIP Return
      L     DB1831.DBD  558;
      T     DB1835.DBD  186;
      L     DB1835.DBD  138;
      T     DB1831.DBD  562;

//CIP Prerun
      L     DB1831.DBD  542;
      T     DB1835.DBD  190;
      L     DB1835.DBD  142;
      T     DB1831.DBD  546;

// Write Own Data to CIP
      L     DB1835.DBD   10;
      T     DB1835.DBD  154;

      L     DB1835.DBW   14;
      T     DB1835.DBW  158;

      L     DB1835.DBW   16;
      T     DB1835.DBW  160;

      L     DB1835.DBW   18;
      T     DB1835.DBW  162;

      L     DB1835.DBW   20;
      T     DB1835.DBW  164;

      L     DB1835.DBW   22;
      T     DB1835.DBW  166;

      A     DB1835.DBX   24.0;
      =     DB1835.DBX  168.0;

      A     DB1835.DBX   24.1;
      =     DB1835.DBX  168.1;

      A     DB1835.DBX   24.2;
      =     DB1835.DBX  168.2;

      A     DB1835.DBX   24.3;
      =     DB1835.DBX  168.3;

      A     DB1835.DBX   24.4;
      =     DB1835.DBX  168.4;

      A     DB1835.DBX   24.5;
      =     DB1835.DBX  168.5;

      A     DB1835.DBX   24.6;
      =     DB1835.DBX  168.6;

      A     DB1835.DBX   24.7;
      =     DB1835.DBX  168.7;

// Copy Data to CIP
      CALL SFC   20 (
           SRCBLK                   := DB1835.ToCIP,
           RET_VAL                  := #iRetVal,
           DSTBLK                   := DB1835.ToCIP);

NCIP: NOP   0;

//Empty Signal
      A     DB2831.DBX   78.7;
      =     DB1835.DBX   26.5;

//Full Signal
      AN    DB2831.DBX  138.7;
      O     DB2833.DBX  138.4;
      =     DB1835.DBX   26.2;

//CIP Program Selected
      A     #CIP;
      =     DB1835.DBX   27.1;

// Emergency Stop
      A     #EStopOK; //If needed add or replace with own SpI
      =     DB1835.DBX   27.0; //Emergency Stop OK


NETWORK
TITLE = read from other unit data



END_FUNCTION_BLOCK

FUNCTION_BLOCK FB 1839
TITLE =U083: Hot Water Tank
AUTHOR : Woermann
FAMILY : BOTEC_F1
NAME : Sim
VERSION : 0.1


VAR_TEMP
  CIP : BOOL ;	//CIP active
  xTmp : BOOL ;	//Temporary BOOL (free for general use)
  iTmp : INT ;	//Temporary INT (free for general use)
  rTmp : REAL ;	//Temporary REAL (free for general use)
  UnitNo : INT ;	//Unit Number
END_VAR
BEGIN
NETWORK
TITLE =General

      SET   ;
// get unit number ----------------------------------------------------------
      L     DB1830.DBW    0;
      T     #UnitNo;

// CIP ----------------------------------------------------------------------
      L     DB1831.DBD   54;
      L     0;
      <D    ;
      =     #CIP;

NETWORK
TITLE =Actuator

      A     DB1831.DBX   17.3;
      =     DB2830.DBX  105.3;
      =     DB2830.DBX  185.3;
      =     DB2830.DBX  265.3;
      =     DB2830.DBX  345.3;
      =     DB2830.DBX  425.3;
      =     DB2830.DBX  585.3;
      =     DB2830.DBX  745.3;
      =     DB2830.DBX  825.3;
      =     DB2830.DBX  905.3;
      =     DB2830.DBX  985.3;
      =     DB2830.DBX 1065.3;

NETWORK
TITLE =Special Input

      A     DB1831.DBX   17.3;
      =     DB2831.DBX   81.3;
      =     DB2831.DBX  141.3;
      =     DB2831.DBX  201.3;
      =     DB2831.DBX  261.3;
      =     DB2831.DBX  321.3;
      =     DB2831.DBX  381.3;
      =     DB2831.DBX  441.3;

NETWORK
TITLE =Counter

      A     DB1831.DBX   17.3;
      A     M    101.0;
      =     DB2832.DBX   99.1;

      CLR   ;
NETWORK
TITLE =Analog Input

      A     DB1831.DBX   17.3;
      =     DB2833.DBX  141.3;
      =     DB2833.DBX  261.3;
      =     DB2833.DBX  381.3;
      =     DB2833.DBX  501.3;
      =     DB2833.DBX  621.3;
      =     DB2833.DBX  741.3;

NETWORK
TITLE =Universal Value

      A     DB1831.DBX   17.3;
//      =     "U083UnVD".unv001.Sim;
//      =     "U083UnVD".unv002.Sim;

NETWORK
TITLE =PID

      A     DB1831.DBX   17.3;
//      =     "U083PIDD".HWP1_FU.Ign;
//      =     "U083PIDD".RV_Kaltwasser.Ign;

NETWORK
TITLE =Message

      A     DB1831.DBX   17.3;
//      =     "U083MsgD".msg001.Sim;
//      =     "U083MsgD".msg002.Sim;

NETWORK
TITLE =VLT

      A     DB1831.DBX   17.3;

END_FUNCTION_BLOCK

FUNCTION_BLOCK FB 1845
TITLE =U084: Fresh Water Tank
FAMILY : BOTEC_F1
NAME : Comm
VERSION : 0.1


VAR_TEMP
  iRetVal : INT ;	//return value as integer
  wRetVal : WORD ;	//return value as word
  Run : BOOL ;	//Unit in "RUN" mode
  EStopOK : BOOL ;	//Emergency Stop OK
  CIP : BOOL ;	//CIP Program Selected
  ComCIP : BOOL ;	//Communication with CIP Active
  xTmp : BOOL ;	//Temporary BOOL (free for general use)
  iTmp : INT ;	//Temporary INT (free for general use)
  rTmp : REAL ;	//Temporary REAL (free for general use)
  dTmp : DINT ;	//Temporary DINT (free for general use)
  UnitNo : INT ;	//Unit Number
  EquipmentID : INT ;	//Equipment ID
  Prid : DINT ;	//Process ID
  SFM36 : STRUCT 	// CIP Pump Mode
   I00 : BOOL ;	// Off
   I01 : BOOL ;	// Flow
   I02 : BOOL ;	// Pressure
   I03 : BOOL ;	// Fix Speed
   I04 : BOOL ;
   I05 : BOOL ;
   I06 : BOOL ;
   I07 : BOOL ;
   I08 : BOOL ;
   I09 : BOOL ;
   I10 : BOOL ;
   I11 : BOOL ;
   I12 : BOOL ;
   I13 : BOOL ;
   I14 : BOOL ;
   I15 : BOOL ;
   I16 : BOOL ;
   I17 : BOOL ;
   I18 : BOOL ;
   I19 : BOOL ;
   I20 : BOOL ;
   I21 : BOOL ;
   I22 : BOOL ;
   I23 : BOOL ;
   I24 : BOOL ;
   I25 : BOOL ;
   I26 : BOOL ;
   I27 : BOOL ;
   I28 : BOOL ;
   I29 : BOOL ;
   I30 : BOOL ;
   I31 : BOOL ;
  END_STRUCT ;
END_VAR
BEGIN
NETWORK
TITLE =general

      SET   ;

// unit & equipment number ---------------------------------------------------
      L     DB1840.DBW    0;
      T     #UnitNo;

      L     DB1845.DBW   14;
      L     1000;
      *I    ;
      L     #UnitNo;
      +I    ;
      T     #EquipmentID;

// CIP ----------------------------------------------------------------------
      L     DB1845.DBW   18;
      L     0;
      <I    ;
      =     #CIP;

// Communicating Units-------------------------------------------------------
      L     DB1845.DBD   10;
      L     DB1845.DBD  106;
      ==D   ;
      =     #ComCIP;

// emergency OK -------------------------------------------------------------
      A     DB1845.DBX   75.0; //General Emergency Stop OK
      =     #EStopOK;

NETWORK
TITLE =read other unit's data

      SET   ;

// ... General Unit ----------/

      CALL FC   563 (
           ActReq                   := M    101.0,
           PLCNo                    := DB1845.DBW   14,
           SourceUnitNo             := 99,
           IsTUnit                  := FALSE,
           DstComDRec               := DB1845.GEN,
           RET_VAL                  := #wRetVal);

NETWORK
TITLE =remote start

      SET   ;

      A     DB1841.DBX   15.0;
      A     DB1841.DBX   17.4;
      JCN   Strt;
      L     DB1845.DBD   10;
      L     L#-1; // Prid negative to start on its own
      T     #Prid;

      CALL FC    48 (
           UnitNo                   := #UnitNo,
           PrId                     := #Prid,
           Run                      := DB1841.DBX   17.4,
           PrIdTransfer             := TRUE,
           Start                    := TRUE,
           RetVal                   := #wRetVal);
Strt: NOP   0;
NETWORK
TITLE =external releases

      SET   ;
      =     DB2840.DBX  186.7;
      =     DB2840.DBX  666.7;
      =     DB2840.DBX  746.7;
NETWORK
TITLE =write own unit data

      SET   ;

//-- CIP Communication ---------------------------------------
      AN    DB1841.DBX   15.0;
//      AN "U084SeqD".Seq.PO.B30 // CIP Active (Slave)
      A     #ComCIP;
      JCN   NCIP;
//Conductivity CIP Return
      L     DB1845.DBD  150;
      T     DB1841.DBD  626;

//Temperature CIP Return
      L     DB1845.DBD  146;
      T     DB1841.DBD  594;

//CIP Prerun Pump SP

      CALL FC    45 (
           SFM                      := DB1841.DBD  686,
           Indexes                  := #SFM36);


      L     0.000000e+000;
      A     #SFM36.I01;
      =     DB1845.DBX  171.7;
      JCN   pfc;
      L     DB1841.DBD  654;
pfc:  NOP   0;
      A     #SFM36.I02;
      =     DB1845.DBX  172.0;
      JCN   ppc;
      L     DB1841.DBD  670;
ppc:  NOP   0;
      A     #SFM36.I03;
      =     DB1845.DBX  171.6;
      JCN   pxc;
      L     DB1841.DBD  574;
pxc:  NOP   0;
      T     DB1845.DBD  182;

//CIP Return
      L     DB1841.DBD  558;
      T     DB1845.DBD  186;
      L     DB1845.DBD  138;
      T     DB1841.DBD  562;

//CIP Prerun
      L     DB1841.DBD  542;
      T     DB1845.DBD  190;
      L     DB1845.DBD  142;
      T     DB1841.DBD  546;

// Write Own Data to CIP
      L     DB1845.DBD   10;
      T     DB1845.DBD  154;

      L     DB1845.DBW   14;
      T     DB1845.DBW  158;

      L     DB1845.DBW   16;
      T     DB1845.DBW  160;

      L     DB1845.DBW   18;
      T     DB1845.DBW  162;

      L     DB1845.DBW   20;
      T     DB1845.DBW  164;

      L     DB1845.DBW   22;
      T     DB1845.DBW  166;

      A     DB1845.DBX   24.0;
      =     DB1845.DBX  168.0;

      A     DB1845.DBX   24.1;
      =     DB1845.DBX  168.1;

      A     DB1845.DBX   24.2;
      =     DB1845.DBX  168.2;

      A     DB1845.DBX   24.3;
      =     DB1845.DBX  168.3;

      A     DB1845.DBX   24.4;
      =     DB1845.DBX  168.4;

      A     DB1845.DBX   24.5;
      =     DB1845.DBX  168.5;

      A     DB1845.DBX   24.6;
      =     DB1845.DBX  168.6;

      A     DB1845.DBX   24.7;
      =     DB1845.DBX  168.7;

// Copy Data to CIP
      CALL SFC   20 (
           SRCBLK                   := DB1845.ToCIP,
           RET_VAL                  := #iRetVal,
           DSTBLK                   := DB1845.ToCIP);

NCIP: NOP   0;

//Empty Signal
      A     DB2841.DBX   78.7;
      =     DB1845.DBX   26.5;

//Full Signal
      AN    DB2841.DBX  138.7;
      O     DB2843.DBX  138.4;
      =     DB1845.DBX   26.2;

//CIP Program Selected
      A     #CIP;
      =     DB1845.DBX   27.1;

// Emergency Stop
      A     #EStopOK; //If needed add or replace with own SpI
      =     DB1845.DBX   27.0; //Emergency Stop OK


NETWORK
TITLE = read from other unit data



END_FUNCTION_BLOCK

FUNCTION_BLOCK FB 1849
TITLE =U084: Fresh Water Tank
AUTHOR : Woermann
FAMILY : BOTEC_F1
NAME : Sim
VERSION : 0.1


VAR_TEMP
  CIP : BOOL ;	//CIP active
  xTmp : BOOL ;	//Temporary BOOL (free for general use)
  iTmp : INT ;	//Temporary INT (free for general use)
  rTmp : REAL ;	//Temporary REAL (free for general use)
  UnitNo : INT ;	//Unit Number
END_VAR
BEGIN
NETWORK
TITLE =General

      SET   ;
// get unit number ----------------------------------------------------------
      L     DB1840.DBW    0;
      T     #UnitNo;

// CIP ----------------------------------------------------------------------
      L     DB1841.DBD   54;
      L     0;
      <D    ;
      =     #CIP;

NETWORK
TITLE =Actuator

      A     DB1841.DBX   17.3;
      =     DB2840.DBX  185.3;
      =     DB2840.DBX  665.3;
      =     DB2840.DBX  745.3;

NETWORK
TITLE =Special Input

      A     DB1841.DBX   17.3;
      =     DB2841.DBX   81.3;
      =     DB2841.DBX  141.3;
      =     DB2841.DBX  201.3;
      =     DB2841.DBX  321.3;
      =     DB2841.DBX  381.3;
      =     DB2841.DBX  441.3;
      =     DB2841.DBX  501.3;
      =     DB2841.DBX  621.3;
      =     DB2841.DBX  681.3;
      =     DB2841.DBX  741.3;
      =     DB2841.DBX  921.3;

NETWORK
TITLE =Counter

      A     DB1841.DBX   17.3;
      A     M    101.0;


      CLR   ;
NETWORK
TITLE =Analog Input

      A     DB1841.DBX   17.3;
      =     DB2843.DBX  141.3;

NETWORK
TITLE =Universal Value

      A     DB1841.DBX   17.3;
//      =     "U084UnVD".unv001.Sim;
//      =     "U084UnVD".unv002.Sim;

NETWORK
TITLE =PID

      A     DB1841.DBX   17.3;

NETWORK
TITLE =Message

      A     DB1841.DBX   17.3;
//      =     "U084MsgD".msg001.Sim;
//      =     "U084MsgD".msg002.Sim;

NETWORK
TITLE =VLT

      A     DB1841.DBX   17.3;

END_FUNCTION_BLOCK

FUNCTION_BLOCK FB 1915
TITLE =U091: CIP Line 1
FAMILY : BOTEC_F1
NAME : Comm
VERSION : 0.1


VAR_TEMP
  iRetVal : INT ;	//return value as integer
  wRetVal : WORD ;	//return value as word
  Run : BOOL ;	//Unit in "RUN" mode
  EStopOK : BOOL ;	//Emergency Stop OK
  CIP : BOOL ;	//CIP Program Selected
  ComCIP : BOOL ;	//Communication with CIP Active
  xTmp : BOOL ;	//Temporary BOOL (free for general use)
  iTmp : INT ;	//Temporary INT (free for general use)
  rTmp : REAL ;	//Temporary REAL (free for general use)
  dTmp : DINT ;	//Temporary DINT (free for general use)
  UnitNo : INT ;	//Unit Number
  EquipmentID : INT ;	//Equipment ID
  Prid : DINT ;	//Process ID
  SFM36 : STRUCT 	// CIP Pump Mode
   I00 : BOOL ;	// Off
   I01 : BOOL ;	// Flow
   I02 : BOOL ;	// Pressure
   I03 : BOOL ;	// Fix Speed
   I04 : BOOL ;
   I05 : BOOL ;
   I06 : BOOL ;
   I07 : BOOL ;
   I08 : BOOL ;
   I09 : BOOL ;
   I10 : BOOL ;
   I11 : BOOL ;
   I12 : BOOL ;
   I13 : BOOL ;
   I14 : BOOL ;
   I15 : BOOL ;
   I16 : BOOL ;
   I17 : BOOL ;
   I18 : BOOL ;
   I19 : BOOL ;
   I20 : BOOL ;
   I21 : BOOL ;
   I22 : BOOL ;
   I23 : BOOL ;
   I24 : BOOL ;
   I25 : BOOL ;
   I26 : BOOL ;
   I27 : BOOL ;
   I28 : BOOL ;
   I29 : BOOL ;
   I30 : BOOL ;
   I31 : BOOL ;
  END_STRUCT ;
END_VAR
BEGIN
NETWORK
TITLE =general

      SET   ;

// unit & equipment number ---------------------------------------------------
      L     DB1910.DBW    0;
      T     #UnitNo;

      L     DB1915.DBW   14;
      L     1000;
      *I    ;
      L     #UnitNo;
      +I    ;
      T     #EquipmentID;

// CIP ----------------------------------------------------------------------
      L     DB1915.DBW   18;
      L     0;
      <I    ;
      =     #CIP;

// Communicating Units-------------------------------------------------------
      L     DB1915.DBD   10;
      L     DB1915.DBD  106;
      ==D   ;
      =     #ComCIP;

// emergency OK -------------------------------------------------------------
      A     DB1915.DBX   75.0; //General Emergency Stop OK
      =     #EStopOK;

NETWORK
TITLE =remote start

      SET   ;
      L     DB502.DBD    0;
      L     0;
      >D    ;
      A     DB1911.DBX   15.0;
      A     DB1911.DBX   17.4;
      JCN   Strt;
      L     DB502.DBD    0;
      T     #Prid;

      CALL FC    48 (
           UnitNo                   := #UnitNo,
           PrId                     := #Prid,
           Run                      := DB1911.DBX   17.4,
           PrIdTransfer             := TRUE,
           Start                    := TRUE,
           RetVal                   := #wRetVal);
Strt: NOP   0;

      L     0;
      T     DB502.DBD    0; // Reset Start Request

END_FUNCTION_BLOCK

FUNCTION_BLOCK FB 1919
TITLE =U091: CIP Line 1
AUTHOR : Woermann
FAMILY : BOTEC_F1
NAME : Sim
VERSION : 0.1


VAR_TEMP
  CIP : BOOL ;	//CIP active
  xTmp : BOOL ;	//Temporary BOOL (free for general use)
  iTmp : INT ;	//Temporary INT (free for general use)
  rTmp : REAL ;	//Temporary REAL (free for general use)
  UnitNo : INT ;	//Unit Number
END_VAR
BEGIN
NETWORK
TITLE =General

      SET   ;
// get unit number ----------------------------------------------------------
      L     DB1910.DBW    0;
      T     #UnitNo;

// CIP ----------------------------------------------------------------------
      L     DB1911.DBD   54;
      L     0;
      <D    ;
      =     #CIP;

NETWORK
TITLE =Actuator
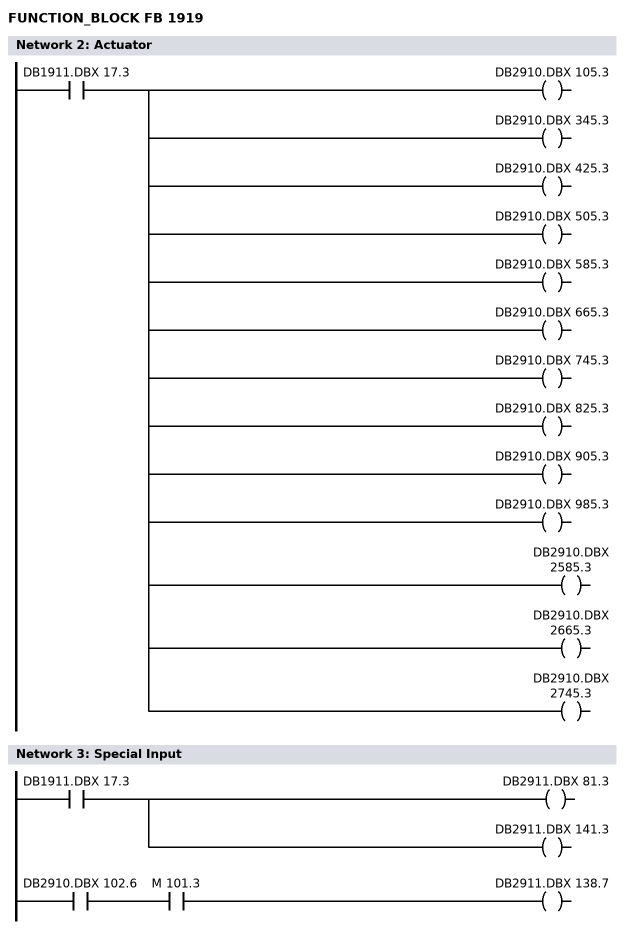

      A     DB1911.DBX   17.3;
      =     DB2910.DBX  105.3;
      =     DB2910.DBX  345.3;
      =     DB2910.DBX  425.3;
      =     DB2910.DBX  505.3;
      =     DB2910.DBX  585.3;
      =     DB2910.DBX  665.3;
      =     DB2910.DBX  745.3;
      =     DB2910.DBX  825.3;
      =     DB2910.DBX  905.3;
      =     DB2910.DBX  985.3;
      =     DB2910.DBX 2585.3;
      =     DB2910.DBX 2665.3;
      =     DB2910.DBX 2745.3;

NETWORK
TITLE =Special Input

      A     DB1911.DBX   17.3;
      =     DB2911.DBX   81.3;
      =     DB2911.DBX  141.3;

      A     DB2910.DBX  102.6;
      A     M    101.3;
      =     DB2911.DBX  138.7;

NETWORK
TITLE =Counter

      A     DB1911.DBX   17.3;
//      =     "U091CntD".IDM_IMPULSE_RV_1FQI.Sim;
      A     M    101.0;
      =     DB2912.DBX  179.1;
      CLR   ;
NETWORK
TITLE =Analog Input

      A     DB1911.DBX   17.3;
      =     DB2913.DBX  141.3;
      =     DB2913.DBX  261.3;
      =     DB2913.DBX  381.3;
      =     DB2913.DBX  501.3;

NETWORK
TITLE =Universal Value

      A     DB1911.DBX   17.3;
//      =     "U091UnVD".unv001.Sim;
//      =     "U091UnVD".unv002.Sim;

NETWORK
TITLE =PID

      A     DB1911.DBX   17.3;
//      =     "U091PIDD".RV1RV.Ign;

NETWORK
TITLE =Message

      A     DB1911.DBX   17.3;
//      =     "U091MsgD".msg001.Sim;
//      =     "U091MsgD".msg002.Sim;

NETWORK
TITLE =VLT

      A     DB1911.DBX   17.3;

END_FUNCTION_BLOCK

FUNCTION_BLOCK FB 1925
TITLE =U092: CIP Line 2
FAMILY : BOTEC_F1
NAME : Comm
VERSION : 0.1


VAR_TEMP
  iRetVal : INT ;	//return value as integer
  wRetVal : WORD ;	//return value as word
  Run : BOOL ;	//Unit in "RUN" mode
  EStopOK : BOOL ;	//Emergency Stop OK
  CIP : BOOL ;	//CIP Program Selected
  ComCIP : BOOL ;	//Communication with CIP Active
  xTmp : BOOL ;	//Temporary BOOL (free for general use)
  iTmp : INT ;	//Temporary INT (free for general use)
  rTmp : REAL ;	//Temporary REAL (free for general use)
  dTmp : DINT ;	//Temporary DINT (free for general use)
  UnitNo : INT ;	//Unit Number
  EquipmentID : INT ;	//Equipment ID
  Prid : DINT ;	//Process ID
  SFM36 : STRUCT 	// CIP Pump Mode
   I00 : BOOL ;	// Off
   I01 : BOOL ;	// Flow
   I02 : BOOL ;	// Pressure
   I03 : BOOL ;	// Fix Speed
   I04 : BOOL ;
   I05 : BOOL ;
   I06 : BOOL ;
   I07 : BOOL ;
   I08 : BOOL ;
   I09 : BOOL ;
   I10 : BOOL ;
   I11 : BOOL ;
   I12 : BOOL ;
   I13 : BOOL ;
   I14 : BOOL ;
   I15 : BOOL ;
   I16 : BOOL ;
   I17 : BOOL ;
   I18 : BOOL ;
   I19 : BOOL ;
   I20 : BOOL ;
   I21 : BOOL ;
   I22 : BOOL ;
   I23 : BOOL ;
   I24 : BOOL ;
   I25 : BOOL ;
   I26 : BOOL ;
   I27 : BOOL ;
   I28 : BOOL ;
   I29 : BOOL ;
   I30 : BOOL ;
   I31 : BOOL ;
  END_STRUCT ;
END_VAR
BEGIN
NETWORK
TITLE =general

      SET   ;

// unit & equipment number ---------------------------------------------------
      L     DB1920.DBW    0;
      T     #UnitNo;

      L     DB1925.DBW   14;
      L     1000;
      *I    ;
      L     #UnitNo;
      +I    ;
      T     #EquipmentID;

// CIP ----------------------------------------------------------------------
      L     DB1925.DBW   18;
      L     0;
      <I    ;
      =     #CIP;

// Communicating Units-------------------------------------------------------
      L     DB1925.DBD   10;
      L     DB1925.DBD  106;
      ==D   ;
      =     #ComCIP;

// emergency OK -------------------------------------------------------------
      A     DB1925.DBX   75.0; //General Emergency Stop OK
      =     #EStopOK;

NETWORK
TITLE =remote start

      SET   ;
      L     DB502.DBD    4;
      L     0;
      >D    ;
      A     DB1921.DBX   15.0;
      A     DB1921.DBX   17.4;
      JCN   Strt;
      L     DB502.DBD    4;
      T     #Prid;

      CALL FC    48 (
           UnitNo                   := #UnitNo,
           PrId                     := #Prid,
           Run                      := DB1921.DBX   17.4,
           PrIdTransfer             := TRUE,
           Start                    := TRUE,
           RetVal                   := #wRetVal);
Strt: NOP   0;

      L     0;
      T     DB502.DBD    4; // Reset Start Request

END_FUNCTION_BLOCK

FUNCTION_BLOCK FB 1929
TITLE =U092: CIP Line 2
AUTHOR : Woermann
FAMILY : BOTEC_F1
NAME : Sim
VERSION : 0.1


VAR_TEMP
  CIP : BOOL ;	//CIP active
  xTmp : BOOL ;	//Temporary BOOL (free for general use)
  iTmp : INT ;	//Temporary INT (free for general use)
  rTmp : REAL ;	//Temporary REAL (free for general use)
  UnitNo : INT ;	//Unit Number
END_VAR
BEGIN
NETWORK
TITLE =General

      SET   ;
// get unit number ----------------------------------------------------------
      L     DB1920.DBW    0;
      T     #UnitNo;

// CIP ----------------------------------------------------------------------
      L     DB1921.DBD   54;
      L     0;
      <D    ;
      =     #CIP;

NETWORK
TITLE =Actuator
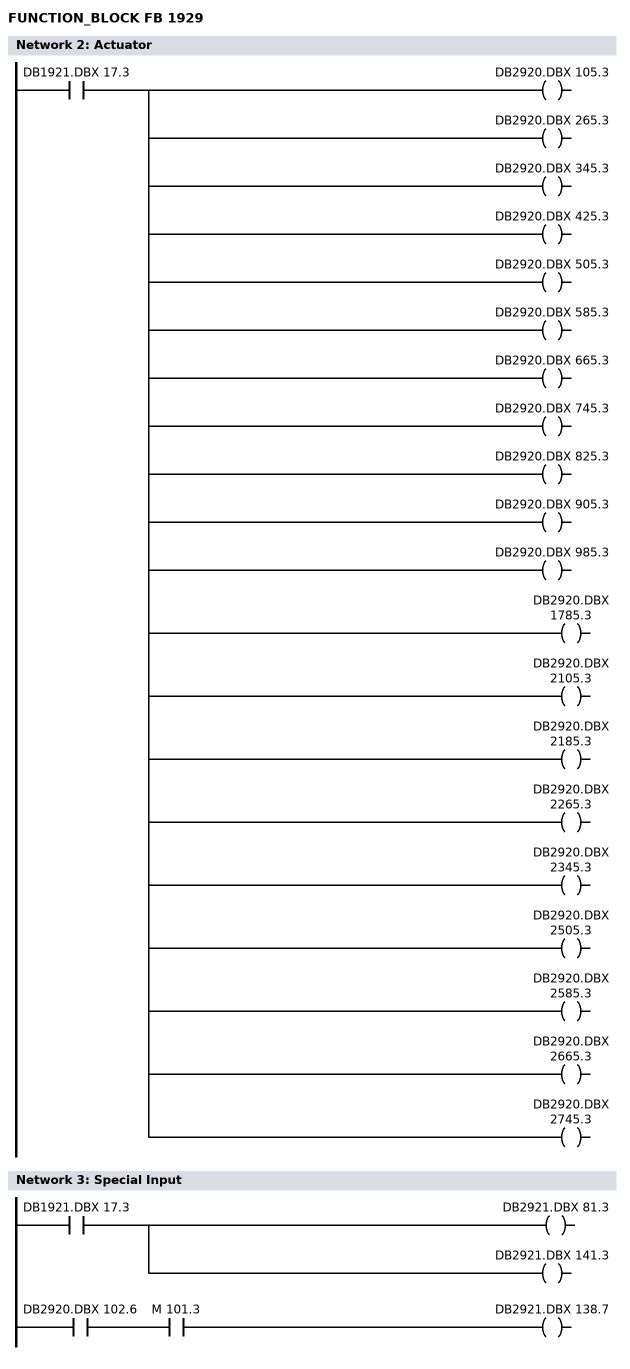

      A     DB1921.DBX   17.3;
      =     DB2920.DBX  105.3;
      =     DB2920.DBX  265.3;
      =     DB2920.DBX  345.3;
      =     DB2920.DBX  425.3;
      =     DB2920.DBX  505.3;
      =     DB2920.DBX  585.3;
      =     DB2920.DBX  665.3;
      =     DB2920.DBX  745.3;
      =     DB2920.DBX  825.3;
      =     DB2920.DBX  905.3;
      =     DB2920.DBX  985.3;
      =     DB2920.DBX 1785.3;
      =     DB2920.DBX 2105.3;
      =     DB2920.DBX 2185.3;
      =     DB2920.DBX 2265.3;
      =     DB2920.DBX 2345.3;
      =     DB2920.DBX 2505.3;
      =     DB2920.DBX 2585.3;
      =     DB2920.DBX 2665.3;
      =     DB2920.DBX 2745.3;


NETWORK
TITLE =Special Input

      A     DB1921.DBX   17.3;
      =     DB2921.DBX   81.3;
      =     DB2921.DBX  141.3;

      A     DB2920.DBX  102.6;
      A     M    101.3;
      =     DB2921.DBX  138.7;

NETWORK
TITLE =Counter

      A     DB1921.DBX   17.3;
//      =     "U092CntD".IDM_IMPULSE_RV_2FQI.Sim;
      A     M    101.0;
      =     DB2922.DBX  179.1;


      CLR   ;
NETWORK
TITLE =Analog Input

      A     DB1921.DBX   17.3;
      =     DB2923.DBX  141.3;
      =     DB2923.DBX  261.3;
      =     DB2923.DBX  381.3;
      =     DB2923.DBX  501.3;

NETWORK
TITLE =Universal Value

      A     DB1921.DBX   17.3;
//      =     "U092UnVD".unv001.Sim;
//      =     "U092UnVD".unv002.Sim;

NETWORK
TITLE =PID

      A     DB1921.DBX   17.3;
//      =     "U092PIDD".RV2RV.Ign;

NETWORK
TITLE =Message

      A     DB1921.DBX   17.3;
//      =     "U092MsgD".msg001.Sim;
//      =     "U092MsgD".msg002.Sim;

NETWORK
TITLE =VLT

      A     DB1921.DBX   17.3;

END_FUNCTION_BLOCK

FUNCTION_BLOCK FB 1935
TITLE =U093: CIP Line 3
FAMILY : BOTEC_F1
NAME : Comm
VERSION : 0.1


VAR_TEMP
  iRetVal : INT ;	//return value as integer
  wRetVal : WORD ;	//return value as word
  Run : BOOL ;	//Unit in "RUN" mode
  EStopOK : BOOL ;	//Emergency Stop OK
  CIP : BOOL ;	//CIP Program Selected
  ComCIP : BOOL ;	//Communication with CIP Active
  xTmp : BOOL ;	//Temporary BOOL (free for general use)
  iTmp : INT ;	//Temporary INT (free for general use)
  rTmp : REAL ;	//Temporary REAL (free for general use)
  dTmp : DINT ;	//Temporary DINT (free for general use)
  UnitNo : INT ;	//Unit Number
  EquipmentID : INT ;	//Equipment ID
  Prid : DINT ;	//Process ID
  SFM36 : STRUCT 	// CIP Pump Mode
   I00 : BOOL ;	// Off
   I01 : BOOL ;	// Flow
   I02 : BOOL ;	// Pressure
   I03 : BOOL ;	// Fix Speed
   I04 : BOOL ;
   I05 : BOOL ;
   I06 : BOOL ;
   I07 : BOOL ;
   I08 : BOOL ;
   I09 : BOOL ;
   I10 : BOOL ;
   I11 : BOOL ;
   I12 : BOOL ;
   I13 : BOOL ;
   I14 : BOOL ;
   I15 : BOOL ;
   I16 : BOOL ;
   I17 : BOOL ;
   I18 : BOOL ;
   I19 : BOOL ;
   I20 : BOOL ;
   I21 : BOOL ;
   I22 : BOOL ;
   I23 : BOOL ;
   I24 : BOOL ;
   I25 : BOOL ;
   I26 : BOOL ;
   I27 : BOOL ;
   I28 : BOOL ;
   I29 : BOOL ;
   I30 : BOOL ;
   I31 : BOOL ;
  END_STRUCT ;
END_VAR
BEGIN
NETWORK
TITLE =general

      SET   ;

// unit & equipment number ---------------------------------------------------
      L     DB1930.DBW    0;
      T     #UnitNo;

      L     DB1935.DBW   14;
      L     1000;
      *I    ;
      L     #UnitNo;
      +I    ;
      T     #EquipmentID;

// CIP ----------------------------------------------------------------------
      L     DB1935.DBW   18;
      L     0;
      <I    ;
      =     #CIP;

// Communicating Units-------------------------------------------------------
      L     DB1935.DBD   10;
      L     DB1935.DBD  106;
      ==D   ;
      =     #ComCIP;

// emergency OK -------------------------------------------------------------
      A     DB1935.DBX   75.0; //General Emergency Stop OK
      =     #EStopOK;

NETWORK
TITLE =remote start

      SET   ;
      L     DB502.DBD    8;
      L     0;
      >D    ;
      A     DB1931.DBX   15.0;
      A     DB1931.DBX   17.4;
      JCN   Strt;
      L     DB502.DBD    8;
      T     #Prid;

      CALL FC    48 (
           UnitNo                   := #UnitNo,
           PrId                     := #Prid,
           Run                      := DB1931.DBX   17.4,
           PrIdTransfer             := TRUE,
           Start                    := TRUE,
           RetVal                   := #wRetVal);
Strt: NOP   0;

      L     0;
      T     DB502.DBD    8; // Reset Start Request


END_FUNCTION_BLOCK

FUNCTION_BLOCK FB 1939
TITLE =U093: CIP Line 3
AUTHOR : Woermann
FAMILY : BOTEC_F1
NAME : Sim
VERSION : 0.1


VAR_TEMP
  CIP : BOOL ;	//CIP active
  xTmp : BOOL ;	//Temporary BOOL (free for general use)
  iTmp : INT ;	//Temporary INT (free for general use)
  rTmp : REAL ;	//Temporary REAL (free for general use)
  UnitNo : INT ;	//Unit Number
END_VAR
BEGIN
NETWORK
TITLE =General

      SET   ;
// get unit number ----------------------------------------------------------
      L     DB1930.DBW    0;
      T     #UnitNo;

// CIP ----------------------------------------------------------------------
      L     DB1931.DBD   54;
      L     0;
      <D    ;
      =     #CIP;

NETWORK
TITLE =Actuator
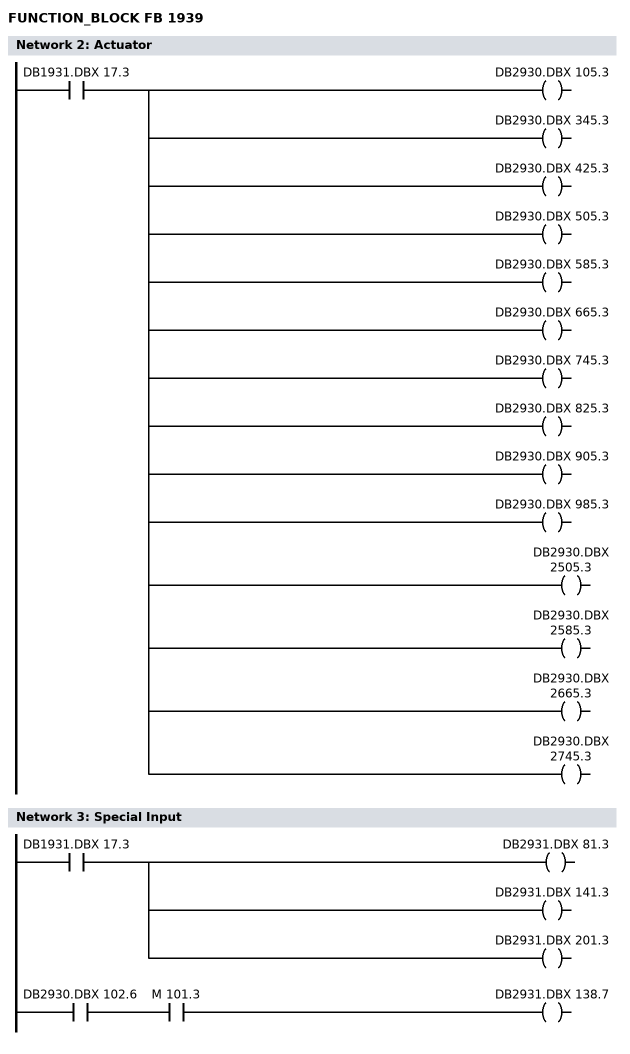

      A     DB1931.DBX   17.3;
      =     DB2930.DBX  105.3;
      =     DB2930.DBX  345.3;
      =     DB2930.DBX  425.3;
      =     DB2930.DBX  505.3;
      =     DB2930.DBX  585.3;
      =     DB2930.DBX  665.3;
      =     DB2930.DBX  745.3;
      =     DB2930.DBX  825.3;
      =     DB2930.DBX  905.3;
      =     DB2930.DBX  985.3;
      =     DB2930.DBX 2505.3;
      =     DB2930.DBX 2585.3;
      =     DB2930.DBX 2665.3;
      =     DB2930.DBX 2745.3;

NETWORK
TITLE =Special Input

      A     DB1931.DBX   17.3;
      =     DB2931.DBX   81.3;
      =     DB2931.DBX  141.3;
      =     DB2931.DBX  201.3;

      A     DB2930.DBX  102.6;
      A     M    101.3;
      =     DB2931.DBX  138.7;

NETWORK
TITLE =Counter

      A     DB1931.DBX   17.3;
//      =     "U093CntD".IDM_IMPULSE_RV_3FQI.Sim;
      A     M    101.0;
      =     DB2932.DBX  179.1;


      CLR   ;
NETWORK
TITLE =Analog Input

      A     DB1931.DBX   17.3;
      =     DB2933.DBX  141.3;
      =     DB2933.DBX  261.3;
      =     DB2933.DBX  381.3;
      =     DB2933.DBX  501.3;

NETWORK
TITLE =Universal Value

      A     DB1931.DBX   17.3;
//      =     "U093UnVD".unv001.Sim;
//      =     "U093UnVD".unv002.Sim;

NETWORK
TITLE =PID

      A     DB1931.DBX   17.3;
//      =     "U093PIDD".RV3RV.Ign;

NETWORK
TITLE =Message

      A     DB1931.DBX   17.3;
//      =     "U093MsgD".msg001.Sim;
//      =     "U093MsgD".msg002.Sim;

NETWORK
TITLE =VLT

      A     DB1931.DBX   17.3;

END_FUNCTION_BLOCK

FUNCTION_BLOCK FB 1945
TITLE =U094: CIP 1 Distribution
FAMILY : BOTEC_F1
NAME : Comm
VERSION : 0.1


VAR_TEMP
  iRetVal : INT ;	//return value as integer
  wRetVal : WORD ;	//return value as word
  Run : BOOL ;	//Unit in "RUN" mode
  EStopOK : BOOL ;	//Emergency Stop OK
  CIP : BOOL ;	//CIP Program Selected
  ComCIP : BOOL ;	//Communication with CIP Active
  xTmp : BOOL ;	//Temporary BOOL (free for general use)
  iTmp : INT ;	//Temporary INT (free for general use)
  rTmp : REAL ;	//Temporary REAL (free for general use)
  dTmp : DINT ;	//Temporary DINT (free for general use)
  UnitNo : INT ;	//Unit Number
  EquipmentID : INT ;	//Equipment ID
  Prid : DINT ;	//Process ID
  SFM36 : STRUCT 	// CIP Pump Mode
   I00 : BOOL ;	// Off
   I01 : BOOL ;	// Flow
   I02 : BOOL ;	// Pressure
   I03 : BOOL ;	// Fix Speed
   I04 : BOOL ;
   I05 : BOOL ;
   I06 : BOOL ;
   I07 : BOOL ;
   I08 : BOOL ;
   I09 : BOOL ;
   I10 : BOOL ;
   I11 : BOOL ;
   I12 : BOOL ;
   I13 : BOOL ;
   I14 : BOOL ;
   I15 : BOOL ;
   I16 : BOOL ;
   I17 : BOOL ;
   I18 : BOOL ;
   I19 : BOOL ;
   I20 : BOOL ;
   I21 : BOOL ;
   I22 : BOOL ;
   I23 : BOOL ;
   I24 : BOOL ;
   I25 : BOOL ;
   I26 : BOOL ;
   I27 : BOOL ;
   I28 : BOOL ;
   I29 : BOOL ;
   I30 : BOOL ;
   I31 : BOOL ;
  END_STRUCT ;
END_VAR
BEGIN
NETWORK
TITLE =general

      SET   ;

// unit & equipment number ---------------------------------------------------
      L     DB1940.DBW    0;
      T     #UnitNo;

      L     DB1945.DBW   14;
      L     1000;
      *I    ;
      L     #UnitNo;
      +I    ;
      T     #EquipmentID;

// CIP ----------------------------------------------------------------------
      L     DB1945.DBW   18;
      L     0;
      <I    ;
      =     #CIP;

// Communicating Units-------------------------------------------------------
      L     DB1945.DBD   10;
      L     DB1945.DBD  106;
      ==D   ;
      =     #ComCIP;

// emergency OK -------------------------------------------------------------
      A     DB1945.DBX   75.0; //General Emergency Stop OK
      =     #EStopOK;

NETWORK
TITLE =read other unit's data

      SET   ;

// ... General Unit ----------/

      CALL FC   563 (
           ActReq                   := M    101.0,
           PLCNo                    := DB1945.DBW   14,
           SourceUnitNo             := 99,
           IsTUnit                  := FALSE,
           DstComDRec               := DB1945.GEN,
           RET_VAL                  := #wRetVal);


// ... CIP Unit ------------- /

      CALL FC   563 (
           ActReq                   := M    101.0,
           PLCNo                    := 3,
           SourceUnitNo             := 91,
           IsTUnit                  := FALSE,
           DstComDRec               := DB1945.CIP,
           RET_VAL                  := #wRetVal);

// ... To CIP Unit ------------- /
      AN    DB1941.DBX   15.0;
      A     DB1941.DBX 1233.6; // CIP Active (Slave)
      O     DB1941.DBX 1230.3; // Production active
//   A     #ComCIP
      JCN   Slav;
      CALL SFC   20 (
           SRCBLK                   := DB502.ToCIP1,
           RET_VAL                  := #iRetVal,
           DSTBLK                   := DB1945.ToCIP);
Slav: NOP   0;

NETWORK
TITLE =remote start

      SET   ;
//-----------------------------------
// Start Request
//-----------------------------------
      L     DB502.DBD  156;
      L     0;
      >D    ;
      A     DB1941.DBX   15.0;
      A     DB1941.DBX   17.4;
      JCN   Strt;
      L     DB502.DBD  156;
      T     #Prid;

